# B&R Automation Studio project GAT (part 3)

### Alarm.mpalarmxcore - 5PPC2200_AL14_000/mappServices/Alarms/Alarm.mpalarmxcore
```
Element gAlarmXMpLink (Type=mpalarmxcore)
  mapp.AlarmX.Core:
    BySeverity:
      [0]:
        Severity = 1..9
        [0] = Reaction
          Name = Info
      [1]:
        Severity = 10..19
        [0] = Reaction
          Name = Warning
      [2]:
        Severity = 20..29
        [0] = Reaction
          Name = Error
  mapp.AlarmX.Core.Configuration:
    [0]:
      Name = EmergencyStop_0
      Message = {$Alarms/EmergencyStop.0}
      Severity = 29
      Behavior = DiscreteValueMonitoring
        Monitoring:
          MonitoredPV = ::AlarmMgt:SafetyInputs.EmergencyStop[0]
          TriggerValues:
            [0] = 1
    [1]:
      Name = EmergencyStop_1
      Message = {$Alarms/EmergencyStop.1}
      Behavior = DiscreteValueMonitoring
        Monitoring:
          MonitoredPV = ::AlarmMgt:SafetyInputs.EmergencyStop[1]
          TriggerValues:
            [0] = 1
    [2]:
      Name = EmergencyStop_2
      Message = {$Alarms/EmergencyStop.2}
      Behavior = DiscreteValueMonitoring
        Monitoring:
          MonitoredPV = ::AlarmMgt:SafetyInputs.EmergencyStop[2]
          TriggerValues:
            [0] = 1
    [3]:
      Name = SafetyDoor_0
      Message = {$Alarms/SafetyDoor.0}
      Severity = 29
      Behavior = DiscreteValueMonitoring
        Monitoring:
          MonitoredPV = ::AlarmMgt:SafetyInputs.SafetyDoor[0]
          TriggerValues:
            [0] = 1
    [4]:
      Name = SafetyDoor_1
      Message = {$Alarms/SafetyDoor.1}
      Severity = 29
      Behavior = DiscreteValueMonitoring
        Monitoring:
          MonitoredPV = ::AlarmMgt:SafetyInputs.SafetyDoor[1]
          TriggerValues:
            [0] = 1
    [5]:
      Name = SafetyDoor_2
      Message = {$Alarms/SafetyDoor.2}
      Severity = 29
      Behavior = DiscreteValueMonitoring
        Monitoring:
          MonitoredPV = ::AlarmMgt:SafetyInputs.SafetyDoor[2]
          TriggerValues:
            [0] = 1
    [6]:
      Name = SafetyDoor_3
      Message = {$Alarms/SafetyDoor.3}
      Severity = 29
      Behavior = DiscreteValueMonitoring
        Monitoring:
          MonitoredPV = ::AlarmMgt:SafetyInputs.SafetyDoor[3]
          TriggerValues:
            [0] = 1
    [7]:
      Name = SafetyDoor_4
      Message = {$Alarms/SafetyDoor.4}
      Severity = 29
      Behavior = DiscreteValueMonitoring
        Monitoring:
          MonitoredPV = ::AlarmMgt:SafetyInputs.SafetyDoor[4]
          TriggerValues:
            [0] = 1
    [8]:
      Name = SafetyDoor_5
      Message = {$Alarms/SafetyDoor.5}
      Severity = 29
      Behavior = DiscreteValueMonitoring
        Monitoring:
          MonitoredPV = ::AlarmMgt:SafetyInputs.SafetyDoor[5]
          TriggerValues:
            [0] = 1
    [9]:
      Name = LevelMonitoringExample
      Message = {$Alarms/LimitMonitoringExample} {=$Alarms/{$LimitText}}
      Behavior = LevelMonitoring
        Monitoring:
          MonitoredPV = ::AlarmMgt:AlarmExamples.LevelMonitoring
          LowLimitEnable = Static
            Limit = 20
            LimitText = LevelMonitoringAlarmLowTextExample
            LowLowLimitEnable = Static
              Limit = 10
              LimitText = LevelMonitoringAlarmLowLowTextExample
          HighLimitEnable = Static
            Limit = 80
            LimitText = LevelMonitoringAlarmHighTextExample
            HighHighLimitEnable = Static
              Limit = 90
              LimitText = LevelMonitoringAlarmHighHighTextExample
    [10]:
      Name = DeviationMonitoringExample
      Message = {$Alarms/LimitText}
      Behavior = DeviationMonitoring
        Monitoring:
          MonitoredPV = ::AlarmMgt:AlarmExamples.DeviationMonitoring
          SetpointPV = ::AlarmMgt:AlarmExamples.DeviationMonitoringSetpoint
          LowLimitEnable = Static
            Limit = -5
            LimitText = Low limit exceeded
          HighLimitEnable = Static
            Limit = 5
            LimitText = High limit exceeded
    [11]:
      Name = RateOfChangeExample
      Message = {$Alarms/RateOfChangeAlarmExample}
      Behavior = RateOfChangeMonitoring
        Monitoring:
          MonitoredPV = ::AlarmMgt:AlarmExamples.RateOfChange
          HighLimitEnable = Static
            Limit = 5
            LimitText = High limit exceeded
    [12]:
      Name = SnippetExample
      Message = {$Alarms/SnippetAlarmExample}
      Behavior = DiscreteValueMonitoring
        Monitoring:
          MonitoredPV = ::AlarmMgt:AlarmExamples.SnippetValue
          TriggerValues:
            [0] = 50..100
    [13]:
      Name = MpAlarmXControlExample
      Message = {$Alarms/Alarm.0}
      Severity = 20
      Behavior:
        Async = TRUE
    [14]:
      Name = Alarm0
      Message = {$Alarms/Alarm.0}
      Behavior = DiscreteValueMonitoring
        Monitoring:
          MonitoredPV = ::AlarmMgt:Alarms[0]
          InhibitPV = ::AlarmMgt:CommissioningModeActive
          TriggerValues:
            [0] = 1
    [15]:
      Name = Alarm1
      Message = {$Alarms/Alarm.1}
      Code = 1
      Behavior = DiscreteValueMonitoring
        Monitoring:
          MonitoredPV = ::AlarmMgt:Alarms[1]
          TriggerValues:
            [0] = 1
    [16]:
      Name = Alarm2
      Message = {$Alarms/Alarm.2}
      Code = 2
      Behavior = DiscreteValueMonitoring
        Monitoring:
          MonitoredPV = ::AlarmMgt:Alarms[2]
          TriggerValues:
            [0] = 1
    [17]:
      Name = Alarm3
      Message = {$Alarms/Alarm.3}
      Code = 3
      Behavior = DiscreteValueMonitoring
        Monitoring:
          MonitoredPV = ::AlarmMgt:Alarms[3]
          TriggerValues:
            [0] = 1
    [18]:
      Name = Alarm4
      Message = {$Alarms/Alarm.4}
      Code = 4
      Behavior = DiscreteValueMonitoring
        Monitoring:
          MonitoredPV = ::AlarmMgt:Alarms[4]
          TriggerValues:
            [0] = 1
    [19]:
      Name = Alarm5
      Message = {$Alarms/Alarm.5}
      Code = 5
      Behavior = DiscreteValueMonitoring
        Monitoring:
          MonitoredPV = ::AlarmMgt:Alarms[5]
          TriggerValues:
            [0] = 1
    [20]:
      Name = Alarm6
      Message = {$Alarms/Alarm.6}
      Code = 6
      Behavior = DiscreteValueMonitoring
        Monitoring:
          MonitoredPV = ::AlarmMgt:Alarms[6]
          TriggerValues:
            [0] = 1
    [21]:
      Name = Alarm7
      Message = {$Alarms/Alarm.7}
      Code = 7
      Behavior = DiscreteValueMonitoring
        Monitoring:
          MonitoredPV = ::AlarmMgt:Alarms[7]
          TriggerValues:
            [0] = 1
    [22]:
      Name = Alarm8
      Message = {$Alarms/Alarm.8}
      Code = 8
      Behavior = DiscreteValueMonitoring
        Monitoring:
          MonitoredPV = ::AlarmMgt:Alarms[8]
          TriggerValues:
            [0] = 1
    [23]:
      Name = Alarm9
      Message = {$Alarms/Alarm.9}
      Code = 9
      Behavior = DiscreteValueMonitoring
        Monitoring:
          MonitoredPV = ::AlarmMgt:Alarms[9]
          TriggerValues:
            [0] = 1
    [24]:
      Name = Alarm10
      Message = {$Alarms/Alarm.10}
      Code = 10
      Behavior = DiscreteValueMonitoring
        Monitoring:
          MonitoredPV = ::AlarmMgt:Alarms[10]
          TriggerValues:
            [0] = 1
    [25]:
      Name = Alarm11
      Message = {$Alarms/Alarm.11}
      Code = 11
      Behavior = DiscreteValueMonitoring
        Monitoring:
          MonitoredPV = ::AlarmMgt:Alarms[11]
          TriggerValues:
            [0] = 1
    [26]:
      Name = Alarm12
      Message = {$Alarms/Alarm.12}
      Code = 12
      Behavior = DiscreteValueMonitoring
        Monitoring:
          MonitoredPV = ::AlarmMgt:Alarms[12]
          TriggerValues:
            [0] = 1
    [27]:
      Name = Alarm13
      Message = {$Alarms/Alarm.13}
      Code = 13
      Behavior = DiscreteValueMonitoring
        Monitoring:
          MonitoredPV = ::AlarmMgt:Alarms[13]
          TriggerValues:
            [0] = 1
    [28]:
      Name = Alarm14
      Message = {$Alarms/Alarm.14}
      Code = 14
      Behavior = DiscreteValueMonitoring
        Monitoring:
          MonitoredPV = ::AlarmMgt:Alarms[14]
          TriggerValues:
            [0] = 1
    [29]:
      Name = Alarm15
      Message = {$Alarms/Alarm.15}
      Code = 15
      Behavior = DiscreteValueMonitoring
        Monitoring:
          MonitoredPV = ::AlarmMgt:Alarms[15]
          TriggerValues:
            [0] = 1
    [30]:
      Name = Alarm16
      Message = {$Alarms/Alarm.16}
      Code = 16
      Behavior = DiscreteValueMonitoring
        Monitoring:
          MonitoredPV = ::AlarmMgt:Alarms[16]
          TriggerValues:
            [0] = 1
    [31]:
      Name = Alarm17
      Message = {$Alarms/Alarm.17}
      Code = 17
      Behavior = DiscreteValueMonitoring
        Monitoring:
          MonitoredPV = ::AlarmMgt:Alarms[17]
          TriggerValues:
            [0] = 1
    [32]:
      Name = Alarm18
      Message = {$Alarms/Alarm.18}
      Code = 18
      Behavior = DiscreteValueMonitoring
        Monitoring:
          MonitoredPV = ::AlarmMgt:Alarms[18]
          TriggerValues:
            [0] = 1
    [33]:
      Name = Alarm19
      Message = {$Alarms/Alarm.19}
      Code = 19
      Behavior = DiscreteValueMonitoring
        Monitoring:
          MonitoredPV = ::AlarmMgt:Alarms[19]
          TriggerValues:
            [0] = 1
    [34]:
      Name = Alarm20
      Message = {$Alarms/Alarm.20}
      Behavior = DiscreteValueMonitoring
        Monitoring:
          MonitoredPV = ::AlarmMgt:Alarms[20]
          TriggerValues:
            [0] = 1
    [35]:
      Name = Alarm21
      Message = {$Alarms/Alarm.21}
      Code = 21
      Behavior = DiscreteValueMonitoring
        Monitoring:
          MonitoredPV = ::AlarmMgt:Alarms[21]
          TriggerValues:
            [0] = 1
    [36]:
      Name = Alarm22
      Message = {$Alarms/Alarm.22}
      Code = 22
      Behavior = DiscreteValueMonitoring
        Monitoring:
          MonitoredPV = ::AlarmMgt:Alarms[22]
          TriggerValues:
            [0] = 1
    [37]:
      Name = Alarm23
      Message = {$Alarms/Alarm.23}
      Code = 23
      Behavior = DiscreteValueMonitoring
        Monitoring:
          MonitoredPV = ::AlarmMgt:Alarms[23]
          TriggerValues:
            [0] = 1
    [38]:
      Name = Alarm24
      Message = {$Alarms/Alarm.24}
      Code = 24
      Behavior = DiscreteValueMonitoring
        Monitoring:
          MonitoredPV = ::AlarmMgt:Alarms[24]
          TriggerValues:
            [0] = 1
    [39]:
      Name = Alarm25
      Message = {$Alarms/Alarm.25}
      Code = 25
      Behavior = DiscreteValueMonitoring
        Monitoring:
          MonitoredPV = ::AlarmMgt:Alarms[25]
          TriggerValues:
            [0] = 1
    [40]:
      Name = Alarm26
      Message = {$Alarms/Alarm.26}
      Code = 26
      Behavior = DiscreteValueMonitoring
        Monitoring:
          MonitoredPV = ::AlarmMgt:Alarms[26]
          TriggerValues:
            [0] = 1
    [41]:
      Name = Alarm27
      Message = {$Alarms/Alarm.27}
      Code = 27
      Behavior = DiscreteValueMonitoring
        Monitoring:
          MonitoredPV = ::AlarmMgt:Alarms[27]
          TriggerValues:
            [0] = 1
    [42]:
      Name = Alarm28
      Message = {$Alarms/Alarm.28}
      Code = 28
      Behavior = DiscreteValueMonitoring
        Monitoring:
          MonitoredPV = ::AlarmMgt:Alarms[28]
          TriggerValues:
            [0] = 1
    [43]:
      Name = Alarm29
      Message = {$Alarms/Alarm.29}
      Code = 29
      Behavior = DiscreteValueMonitoring
        Monitoring:
          MonitoredPV = ::AlarmMgt:Alarms[29]
          TriggerValues:
            [0] = 1
    [44]:
      Name = Alarm30
      Message = {$Alarms/Alarm.30}
      Behavior = DiscreteValueMonitoring
        Monitoring:
          MonitoredPV = ::AlarmMgt:Alarms[30]
          TriggerValues:
            [0] = 1
    [45]:
      Name = Alarm31
      Message = {$Alarms/Alarm.31}
      Code = 31
      Behavior = DiscreteValueMonitoring
        Monitoring:
          MonitoredPV = ::AlarmMgt:Alarms[31]
          TriggerValues:
            [0] = 1
    [46]:
      Name = Alarm32
      Message = {$Alarms/Alarm.32}
      Code = 32
      Behavior = DiscreteValueMonitoring
        Monitoring:
          MonitoredPV = ::AlarmMgt:Alarms[32]
          TriggerValues:
            [0] = 1
    [47]:
      Name = Alarm33
      Message = {$Alarms/Alarm.33}
      Code = 33
      Behavior = DiscreteValueMonitoring
        Monitoring:
          MonitoredPV = ::AlarmMgt:Alarms[33]
          TriggerValues:
            [0] = 1
    [48]:
      Name = Alarm34
      Message = {$Alarms/Alarm.34}
      Code = 34
      Behavior = DiscreteValueMonitoring
        Monitoring:
          MonitoredPV = ::AlarmMgt:Alarms[34]
          TriggerValues:
            [0] = 1
    [49]:
      Name = Alarm35
      Message = {$Alarms/Alarm.35}
      Code = 35
      Behavior = DiscreteValueMonitoring
        Monitoring:
          MonitoredPV = ::AlarmMgt:Alarms[35]
          TriggerValues:
            [0] = 1
    [50]:
      Name = Alarm36
      Message = {$Alarms/Alarm.36}
      Code = 36
      Behavior = DiscreteValueMonitoring
        Monitoring:
          MonitoredPV = ::AlarmMgt:Alarms[36]
          TriggerValues:
            [0] = 1
    [51]:
      Name = Alarm37
      Message = {$Alarms/Alarm.37}
      Code = 37
      Behavior = DiscreteValueMonitoring
        Monitoring:
          MonitoredPV = ::AlarmMgt:Alarms[37]
          TriggerValues:
            [0] = 1
    [52]:
      Name = Alarm38
      Message = {$Alarms/Alarm.38}
      Code = 38
      Behavior = DiscreteValueMonitoring
        Monitoring:
          MonitoredPV = ::AlarmMgt:Alarms[38]
          TriggerValues:
            [0] = 1
    [53]:
      Name = Alarm39
      Message = {$Alarms/Alarm.39}
      Code = 39
      Behavior = DiscreteValueMonitoring
        Monitoring:
          MonitoredPV = ::AlarmMgt:Alarms[39]
          TriggerValues:
            [0] = 1
    [54]:
      Name = Alarm40
      Message = {$Alarms/Alarm.40}
      Behavior = DiscreteValueMonitoring
        Monitoring:
          MonitoredPV = ::AlarmMgt:Alarms[40]
          TriggerValues:
            [0] = 1
    [55]:
      Name = Alarm41
      Message = {$Alarms/Alarm.41}
      Code = 41
      Behavior = DiscreteValueMonitoring
        Monitoring:
          MonitoredPV = ::AlarmMgt:Alarms[41]
          TriggerValues:
            [0] = 1
    [56]:
      Name = Alarm42
      Message = {$Alarms/Alarm.42}
      Code = 42
      Behavior = DiscreteValueMonitoring
        Monitoring:
          MonitoredPV = ::AlarmMgt:Alarms[42]
          TriggerValues:
            [0] = 1
    [57]:
      Name = Alarm43
      Message = {$Alarms/Alarm.43}
      Code = 43
      Behavior = DiscreteValueMonitoring
        Monitoring:
          MonitoredPV = ::AlarmMgt:Alarms[43]
          TriggerValues:
            [0] = 1
    [58]:
      Name = Alarm44
      Message = {$Alarms/Alarm.44}
      Code = 44
      Behavior = DiscreteValueMonitoring
        Monitoring:
          MonitoredPV = ::AlarmMgt:Alarms[44]
          TriggerValues:
            [0] = 1
    [59]:
      Name = Alarm45
      Message = {$Alarms/Alarm.45}
      Code = 45
      Behavior = DiscreteValueMonitoring
        Monitoring:
          MonitoredPV = ::AlarmMgt:Alarms[45]
          TriggerValues:
            [0] = 1
    [60]:
      Name = Alarm46
      Message = {$Alarms/Alarm.46}
      Code = 46
      Behavior = DiscreteValueMonitoring
        Monitoring:
          MonitoredPV = ::AlarmMgt:Alarms[46]
          TriggerValues:
            [0] = 1
    [61]:
      Name = Alarm47
      Message = {$Alarms/Alarm.47}
      Code = 47
      Behavior = DiscreteValueMonitoring
        Monitoring:
          MonitoredPV = ::AlarmMgt:Alarms[47]
          TriggerValues:
            [0] = 1
    [62]:
      Name = Alarm48
      Message = {$Alarms/Alarm.48}
      Code = 48
      Behavior = DiscreteValueMonitoring
        Monitoring:
          MonitoredPV = ::AlarmMgt:Alarms[48]
          TriggerValues:
            [0] = 1
    [63]:
      Name = Alarm49
      Message = {$Alarms/Alarm.49}
      Code = 49
      Behavior = DiscreteValueMonitoring
        Monitoring:
          MonitoredPV = ::AlarmMgt:Alarms[49]
          TriggerValues:
            [0] = 1
    [64]:
      Name = Alarm50
      Message = {$Alarms/Alarm.50}
      Behavior = DiscreteValueMonitoring
        Monitoring:
          MonitoredPV = ::AlarmMgt:Alarms[50]
          TriggerValues:
            [0] = 1
    [65]:
      Name = Alarm51
      Message = {$Alarms/Alarm.51}
      Code = 51
      Behavior = DiscreteValueMonitoring
        Monitoring:
          MonitoredPV = ::AlarmMgt:Alarms[51]
          TriggerValues:
            [0] = 1
    [66]:
      Name = Alarm52
      Message = {$Alarms/Alarm.52}
      Code = 52
      Behavior = DiscreteValueMonitoring
        Monitoring:
          MonitoredPV = ::AlarmMgt:Alarms[52]
          TriggerValues:
            [0] = 1
    [67]:
      Name = Alarm53
      Message = {$Alarms/Alarm.53}
      Code = 53
      Behavior = DiscreteValueMonitoring
        Monitoring:
          MonitoredPV = ::AlarmMgt:Alarms[53]
          TriggerValues:
            [0] = 1
    [68]:
      Name = Alarm54
      Message = {$Alarms/Alarm.54}
      Code = 54
      Behavior = DiscreteValueMonitoring
        Monitoring:
          MonitoredPV = ::AlarmMgt:Alarms[54]
          TriggerValues:
            [0] = 1
    [69]:
      Name = Alarm55
      Message = {$Alarms/Alarm.55}
      Code = 55
      Behavior = DiscreteValueMonitoring
        Monitoring:
          MonitoredPV = ::AlarmMgt:Alarms[55]
          TriggerValues:
            [0] = 1
    [70]:
      Name = Alarm56
      Message = {$Alarms/Alarm.56}
      Code = 56
      Behavior = DiscreteValueMonitoring
        Monitoring:
          MonitoredPV = ::AlarmMgt:Alarms[56]
          TriggerValues:
            [0] = 1
    [71]:
      Name = Alarm57
      Message = {$Alarms/Alarm.57}
      Code = 57
      Behavior = DiscreteValueMonitoring
        Monitoring:
          MonitoredPV = ::AlarmMgt:Alarms[57]
          TriggerValues:
            [0] = 1
    [72]:
      Name = Alarm58
      Message = {$Alarms/Alarm.58}
      Code = 58
      Behavior = DiscreteValueMonitoring
        Monitoring:
          MonitoredPV = ::AlarmMgt:Alarms[58]
          TriggerValues:
            [0] = 1
    [73]:
      Name = Alarm59
      Message = {$Alarms/Alarm.59}
      Code = 59
      Behavior = DiscreteValueMonitoring
        Monitoring:
          MonitoredPV = ::AlarmMgt:Alarms[59]
          TriggerValues:
            [0] = 1
    [74]:
      Name = Alarm60
      Message = {$Alarms/Alarm.60}
      Behavior = DiscreteValueMonitoring
        Monitoring:
          MonitoredPV = ::AlarmMgt:Alarms[60]
          TriggerValues:
            [0] = 1
    [75]:
      Name = Alarm61
      Message = {$Alarms/Alarm.61}
      Code = 61
      Behavior = DiscreteValueMonitoring
        Monitoring:
          MonitoredPV = ::AlarmMgt:Alarms[61]
          TriggerValues:
            [0] = 1
    [76]:
      Name = Alarm62
      Message = {$Alarms/Alarm.62}
      Code = 62
      Behavior = DiscreteValueMonitoring
        Monitoring:
          MonitoredPV = ::AlarmMgt:Alarms[62]
          TriggerValues:
            [0] = 1
    [77]:
      Name = Alarm63
      Message = {$Alarms/Alarm.63}
      Code = 63
      Behavior = DiscreteValueMonitoring
        Monitoring:
          MonitoredPV = ::AlarmMgt:Alarms[63]
          TriggerValues:
            [0] = 1
    [78]:
      Name = Alarm64
      Message = {$Alarms/Alarm.64}
      Code = 64
      Behavior = DiscreteValueMonitoring
        Monitoring:
          MonitoredPV = ::AlarmMgt:Alarms[64]
          TriggerValues:
            [0] = 1
    [79]:
      Name = Alarm65
      Message = {$Alarms/Alarm.65}
      Code = 65
      Behavior = DiscreteValueMonitoring
        Monitoring:
          MonitoredPV = ::AlarmMgt:Alarms[65]
          TriggerValues:
            [0] = 1
    [80]:
      Name = Alarm66
      Message = {$Alarms/Alarm.66}
      Code = 66
      Behavior = DiscreteValueMonitoring
        Monitoring:
          MonitoredPV = ::AlarmMgt:Alarms[66]
          TriggerValues:
            [0] = 1
    [81]:
      Name = Alarm67
      Message = {$Alarms/Alarm.67}
      Code = 67
      Behavior = DiscreteValueMonitoring
        Monitoring:
          MonitoredPV = ::AlarmMgt:Alarms[67]
          TriggerValues:
            [0] = 1
    [82]:
      Name = Alarm68
      Message = {$Alarms/Alarm.68}
      Code = 68
      Behavior = DiscreteValueMonitoring
        Monitoring:
          MonitoredPV = ::AlarmMgt:Alarms[68]
          TriggerValues:
            [0] = 1
    [83]:
      Name = Alarm69
      Message = {$Alarms/Alarm.69}
      Code = 69
      Behavior = DiscreteValueMonitoring
        Monitoring:
          MonitoredPV = ::AlarmMgt:Alarms[69]
          TriggerValues:
            [0] = 1
    [84]:
      Name = Alarm70
      Message = {$Alarms/Alarm.70}
      Behavior = DiscreteValueMonitoring
        Monitoring:
          MonitoredPV = ::AlarmMgt:Alarms[70]
          TriggerValues:
            [0] = 1
    [85]:
      Name = Alarm71
      Message = {$Alarms/Alarm.71}
      Code = 71
      Behavior = DiscreteValueMonitoring
        Monitoring:
          MonitoredPV = ::AlarmMgt:Alarms[71]
          TriggerValues:
            [0] = 1
    [86]:
      Name = Alarm72
      Message = {$Alarms/Alarm.72}
      Code = 72
      Behavior = DiscreteValueMonitoring
        Monitoring:
          MonitoredPV = ::AlarmMgt:Alarms[72]
          TriggerValues:
            [0] = 1
    [87]:
      Name = Alarm73
      Message = {$Alarms/Alarm.73}
      Code = 73
      Behavior = DiscreteValueMonitoring
        Monitoring:
          MonitoredPV = ::AlarmMgt:Alarms[73]
          TriggerValues:
            [0] = 1
    [88]:
      Name = Alarm74
      Message = {$Alarms/Alarm.74}
      Code = 74
      Behavior = DiscreteValueMonitoring
        Monitoring:
          MonitoredPV = ::AlarmMgt:Alarms[74]
          TriggerValues:
            [0] = 1
    [89]:
      Name = Alarm75
      Message = {$Alarms/Alarm.75}
      Code = 75
      Behavior = DiscreteValueMonitoring
        Monitoring:
          MonitoredPV = ::AlarmMgt:Alarms[75]
          TriggerValues:
            [0] = 1
    [90]:
      Name = Alarm76
      Message = {$Alarms/Alarm.76}
      Code = 76
      Behavior = DiscreteValueMonitoring
        Monitoring:
          MonitoredPV = ::AlarmMgt:Alarms[76]
          TriggerValues:
            [0] = 1
    [91]:
      Name = Alarm77
      Message = {$Alarms/Alarm.77}
      Code = 77
      Behavior = DiscreteValueMonitoring
        Monitoring:
          MonitoredPV = ::AlarmMgt:Alarms[77]
          TriggerValues:
            [0] = 1
    [92]:
      Name = Alarm78
      Message = {$Alarms/Alarm.78}
      Code = 78
      Behavior = DiscreteValueMonitoring
        Monitoring:
          MonitoredPV = ::AlarmMgt:Alarms[78]
          TriggerValues:
            [0] = 1
    [93]:
      Name = Alarm79
      Message = {$Alarms/Alarm.79}
      Code = 79
      Behavior = DiscreteValueMonitoring
        Monitoring:
          MonitoredPV = ::AlarmMgt:Alarms[79]
          TriggerValues:
            [0] = 1
    [94]:
      Name = Alarm80
      Message = {$Alarms/Alarm.80}
      Behavior = DiscreteValueMonitoring
        Monitoring:
          MonitoredPV = ::AlarmMgt:Alarms[80]
          TriggerValues:
            [0] = 1
    [95]:
      Name = Alarm81
      Message = {$Alarms/Alarm.81}
      Code = 81
      Behavior = DiscreteValueMonitoring
        Monitoring:
          MonitoredPV = ::AlarmMgt:Alarms[81]
          TriggerValues:
            [0] = 1
    [96]:
      Name = Alarm82
      Message = {$Alarms/Alarm.82}
      Code = 82
      Behavior = DiscreteValueMonitoring
        Monitoring:
          MonitoredPV = ::AlarmMgt:Alarms[82]
          TriggerValues:
            [0] = 1
    [97]:
      Name = Alarm83
      Message = {$Alarms/Alarm.83}
      Code = 83
      Behavior = DiscreteValueMonitoring
        Monitoring:
          MonitoredPV = ::AlarmMgt:Alarms[83]
          TriggerValues:
            [0] = 1
    [98]:
      Name = Alarm84
      Message = {$Alarms/Alarm.84}
      Code = 84
      Behavior = DiscreteValueMonitoring
        Monitoring:
          MonitoredPV = ::AlarmMgt:Alarms[84]
          TriggerValues:
            [0] = 1
    [99]:
      Name = Alarm85
      Message = {$Alarms/Alarm.85}
      Code = 85
      Behavior = DiscreteValueMonitoring
        Monitoring:
          MonitoredPV = ::AlarmMgt:Alarms[85]
          TriggerValues:
            [0] = 1
    [100]:
      Name = Alarm86
      Message = {$Alarms/Alarm.86}
      Code = 86
      Behavior = DiscreteValueMonitoring
        Monitoring:
          MonitoredPV = ::AlarmMgt:Alarms[86]
          TriggerValues:
            [0] = 1
    [101]:
      Name = Alarm87
      Message = {$Alarms/Alarm.87}
      Code = 87
      Behavior = DiscreteValueMonitoring
        Monitoring:
          MonitoredPV = ::AlarmMgt:Alarms[87]
          TriggerValues:
            [0] = 1
    [102]:
      Name = Alarm88
      Message = {$Alarms/Alarm.88}
      Code = 88
      Behavior = DiscreteValueMonitoring
        Monitoring:
          MonitoredPV = ::AlarmMgt:Alarms[88]
          TriggerValues:
            [0] = 1
    [103]:
      Name = Alarm89
      Message = {$Alarms/Alarm.89}
      Code = 89
      Behavior = DiscreteValueMonitoring
        Monitoring:
          MonitoredPV = ::AlarmMgt:Alarms[89]
          TriggerValues:
            [0] = 1
    [104]:
      Name = Alarm90
      Message = {$Alarms/Alarm.90}
      Behavior = DiscreteValueMonitoring
        Monitoring:
          MonitoredPV = ::AlarmMgt:Alarms[90]
          TriggerValues:
            [0] = 1
    [105]:
      Name = Alarm91
      Message = {$Alarms/Alarm.91}
      Code = 91
      Behavior = DiscreteValueMonitoring
        Monitoring:
          MonitoredPV = ::AlarmMgt:Alarms[91]
          TriggerValues:
            [0] = 1
    [106]:
      Name = Alarm92
      Message = {$Alarms/Alarm.92}
      Code = 92
      Behavior = DiscreteValueMonitoring
        Monitoring:
          MonitoredPV = ::AlarmMgt:Alarms[92]
          TriggerValues:
            [0] = 1
    [107]:
      Name = Alarm93
      Message = {$Alarms/Alarm.93}
      Code = 93
      Behavior = DiscreteValueMonitoring
        Monitoring:
          MonitoredPV = ::AlarmMgt:Alarms[93]
          TriggerValues:
            [0] = 1
    [108]:
      Name = Alarm94
      Message = {$Alarms/Alarm.94}
      Code = 94
      Behavior = DiscreteValueMonitoring
        Monitoring:
          MonitoredPV = ::AlarmMgt:Alarms[94]
          TriggerValues:
            [0] = 1
    [109]:
      Name = Alarm95
      Message = {$Alarms/Alarm.95}
      Code = 95
      Behavior = DiscreteValueMonitoring
        Monitoring:
          MonitoredPV = ::AlarmMgt:Alarms[95]
          TriggerValues:
            [0] = 1
    [110]:
      Name = Alarm96
      Message = {$Alarms/Alarm.96}
      Code = 96
      Behavior = DiscreteValueMonitoring
        Monitoring:
          MonitoredPV = ::AlarmMgt:Alarms[96]
          TriggerValues:
            [0] = 1
    [111]:
      Name = Alarm97
      Message = {$Alarms/Alarm.97}
      Code = 97
      Behavior = DiscreteValueMonitoring
        Monitoring:
          MonitoredPV = ::AlarmMgt:Alarms[97]
          TriggerValues:
            [0] = 1
    [112]:
      Name = Alarm98
      Message = {$Alarms/Alarm.98}
      Code = 98
      Behavior = DiscreteValueMonitoring
        Monitoring:
          MonitoredPV = ::AlarmMgt:Alarms[98]
          TriggerValues:
            [0] = 1
    [113]:
      Name = Alarm99
      Message = {$Alarms/Alarm.99}
      Code = 99
      Behavior = DiscreteValueMonitoring
        Monitoring:
          MonitoredPV = ::AlarmMgt:Alarms[99]
          TriggerValues:
            [0] = 1
  mapp.AlarmX.Core.Snippets:
    AutoDetect = 1
    [0]:
      Key = snippet1
      Value:
        PV = ::AlarmMgt:AlarmExamples.SnippetValue
  mapp.AlarmX.Core.Queries:
    [0]:
      Name = ActiveAlarms
      Update = ::AlarmMgt:AlarmQuery.ActiveAlarmUpdateCount
      Source:
        SELECT:
          [0]:
            PV = ::AlarmMgt:AlarmQuery.Alarms[].Name
          [1]:
            Column = Message
            PV = ::AlarmMgt:AlarmQuery.Alarms[].Message
          [2]:
            Column = Code
            PV = ::AlarmMgt:AlarmQuery.Alarms[].Code
          [3]:
            Column = Severity
            PV = ::AlarmMgt:AlarmQuery.Alarms[].Severity
          [4]:
            Column = Scope
            PV = ::AlarmMgt:AlarmQuery.Alarms[].Scope
          [5]:
            Column = TimeStamp
            PV = ::AlarmMgt:AlarmQuery.Alarms[].TimeStamp
          [6]:
            Column = AdditionalInformation1
            PV = ::AlarmMgt:AlarmQuery.Alarms[].AdditionalInfo
          [7]:
            Column = StateActive
            PV = ::AlarmMgt:AlarmQuery.Alarms[].Active
          [8]:
            Column = StateAcknowledged
            PV = ::AlarmMgt:AlarmQuery.Alarms[].Acknowledged
```

### Axis1Alm.mpalarmxcore - 5PPC2200_AL14_000/mappServices/AppAxis_1/Axis1Alm.mpalarmxcore
```
Element gMpLinkAlarmXCoreAppAxis_1 (Type=mpalarmxcore)
  mapp.AlarmX.Core:
    BySeverity:
      [0]:
        Severity = 1..9
        [0] = Reaction
          Name = Info
        [1] = Escalate
        [2] = Remain
      [1]:
        Severity = 10..19
        [0] = Reaction
          Name = Warning
        [1] = Escalate
        [2] = Remain
      [2]:
        Severity = 20..29
        [0] = Reaction
          Name = Error
        [1] = Escalate
        [2] = Remain
    Default:
      [0] = Reaction
        Name = Duplicate
      [1] = Escalate
      [2] = Remain
  mapp.AlarmX.Core.Configuration:
    [0]:
      Name = ReferenceRequired
      Message = {$IAT/AppAxis_1/Info/Name} : {$Axis/Alarms/ReferenceRequired}
      Severity = 10
      Behavior = DiscreteValueMonitoring
        Monitoring:
          MonitoredPV = ::AppAxis_1:AxisControl.Status.ReferenceRequired
          TriggerValues:
            [0] = 1
    [1]:
      Name = AppAxis_1SpeedNotSet
      Message = {$IAT/AppAxis_1/Info/Name} : {$Axis/Alarms/AppAxis_1SpeedNotSet}
      Code = 250
      Severity = 20
      Behavior:
        Async = TRUE
  mapp.AlarmX.Core.Snippets:
    [0]:
      Key = AppAxis_1Speed
      Value:
        PV = ::AppAxis_1:AxisControl.Parameters.Velocity
```

### Axis1Grp.mpcomgroup - 5PPC2200_AL14_000/mappServices/AppAxis_1/Axis1Grp.mpcomgroup
```
Element gGroupAppAxis_1 (Type=mpcomgroup)
  Linking:
    Subnodes:
      0 = gAppAxis_1
      1 = gAlarmXCore_AppAxis_1
  Alarms = MpAlarmX
```

### AuditCfg.mpaudittrail - 5PPC2200_AL14_000/mappServices/Audit/AuditCfg.mpaudittrail
```
Element gAuditTrailMpLink (Type=mpaudittrail)
  Audit:
    Events:
      [0] = 19
      [1] = 2
      [2] = 48
      [3] = 18
      [4] = 33
    TextSource = TXT
      Name = 
      OutputFormat = EventLog/Root
    Archive = On
    Export:
      FileType = 2
      Encrypt = FALSE
      PDF:
        DefaultFont = 3
  Alarms = MpAlarmX
```

### AuditFile.mpfilemanagerui - 5PPC2200_AL14_000/mappServices/Audit/AuditFile.mpfilemanagerui
```
Element gMpLinkFileManagerUIAudit (Type=mpfilemanagerui)
  Alarms = MpAlarmX
    mapp.AlarmX.Core.Configuration:
      [0]:
        Message = {$File/Alarms/DeviceNotFound}
      [1]:
        Message = {$File/Alarms/AlreadyExisting}
      [2]:
        Message = {$File/Alarms/FileSystemError}
```

### Backup.mpbackupcore - 5PPC2200_AL14_000/mappServices/Backup/Backup.mpbackupcore
```
Element gMpLinkBackupCore (Type=mpbackupcore)
  Backup:
    AutomaticBackup = Enabled
      Mode = Weekly
      OverwriteOldest = Enabled
        MaximumNumberOfBackups = 5
    AutomaticUpdate = Notify
      DeviceName = mappBackup
  Alarms = MpAlarmX
```

### BackupCfg.mpbackupcore - 5PPC2200_AL14_000/mappServices/Backup/BackupCfg.mpbackupcore
```
Element gMpLinkBackupCore (Type=mpbackupcore)
  Backup:
    AutomaticBackup = Enabled
      Mode = Weekly
      OverwriteOldest = Enabled
        MaximumNumberOfBackups = 5
    AutomaticUpdate = Notify
      DeviceName = mappBackupFiles
  Alarms = MpAlarmX
```

### BackupFile.mpfilemanagerui - 5PPC2200_AL14_000/mappServices/Backup/BackupFile.mpfilemanagerui
```
Element gMpLinkFileManagerUIBackup (Type=mpfilemanagerui)
  Alarms = MpAlarmX
```

### ConvAlm.mpalarmxcore - 5PPC2200_AL14_000/mappServices/Conveyor/ConvAlm.mpalarmxcore
```
Element gAlarmXCore_Conveyor (Type=mpalarmxcore)
  mapp.AlarmX.Core:
    BySeverity:
      [0]:
        Severity = 1..9
        [0] = Reaction
          Name = Info
        [1] = Escalate
        [2] = Remain
      [1]:
        Severity = 10..19
        [0] = Reaction
          Name = Warning
        [1] = Escalate
        [2] = Remain
      [2]:
        Severity = 20..29
        [0] = Reaction
          Name = Error
        [1] = Escalate
        [2] = Remain
    Default:
      [0] = Reaction
        Name = Duplicate
      [1] = Escalate
      [2] = Remain
  mapp.AlarmX.Core.Configuration:
    [0]:
      Name = ReferenceRequired
      Message = {$IAT/Conveyor/Info/Name} : {$Conveyor/Alarms/ReferenceRequired}
      Severity = 10
      Behavior = DiscreteValueMonitoring
        Monitoring:
          MonitoredPV = ::Conveyor:AxisControl.Status.ReferenceRequired
          TriggerValues:
            [0] = 1
    [1]:
      Name = ConveyorSpeedNotSet
      Message = {$IAT/Conveyor/Alarms/ConveyorSpeedNotSet}
      Code = 250
      Severity = 20
      Behavior:
        Async = TRUE
  mapp.AlarmX.Core.Snippets:
    [0]:
      Key = ConveyorSpeed
      Value:
        PV = ::Conveyor:AxisControl.Parameters.Velocity
```

### ConvGrp.mpcomgroup - 5PPC2200_AL14_000/mappServices/Conveyor/ConvGrp.mpcomgroup
```
Element gGroupAppAxis_1 (Type=mpcomgroup)
  Linking:
    Subnodes:
      0 = gAxisAppAxis_1
      1 = gAlarmXCore_AppAxis_1
  Alarms = MpAlarmX
```

### CutterAlm.mpalarmxcore - 5PPC2200_AL14_000/mappServices/CrossCutter/CutterAlm.mpalarmxcore
```
Element gAlarmXCore_Cutter (Type=mpalarmxcore)
  mapp.AlarmX.Core:
    BySeverity:
      [0]:
        Severity = 1..9
        [0] = Reaction
          Name = Info
        [1] = Escalate
        [2] = Remain
      [1]:
        Severity = 10..19
        [0] = Reaction
          Name = Warning
        [1] = Escalate
        [2] = Remain
      [2]:
        Severity = 20..29
        [0] = Reaction
          Name = Error
        [1] = Escalate
        [2] = Remain
    Default:
      [0] = Reaction
        Name = Duplicate
      [1] = Escalate
      [2] = Remain
```

### DataCfg.mpdatarecorder - 5PPC2200_AL14_000/mappServices/Data/DataCfg.mpdatarecorder
```
Element gMpLinkDataRecorder (Type=mpdatarecorder)
  DataRecorder:
    MaxFileSize = 10000
    SaveInterval = 2000
    Format = PDF
      Font = 3
      OwnerPassword = 
      AllowCopy = TRUE
      AllowEdit = TRUE
    UnitDefinition = MeasurementSystemBased
      UnitDisplay = 1
  Alarms = MpAlarmX
```

### DataFile.mpfilemanagerui - 5PPC2200_AL14_000/mappServices/Data/DataFile.mpfilemanagerui
```
Element gMpLinkFileManagerUIData (Type=mpfilemanagerui)
  Alarms = MpAlarmX
    mapp.AlarmX.Core.Configuration:
      [0]:
        Message = {$File/Alarms/DeviceNotFound}
      [1]:
        Message = {$File/Alarms/AlreadyExisting}
      [2]:
        Message = {$File/Alarms/FileSystemError}
```

### FileMgr.mpfilemanagerui - 5PPC2200_AL14_000/mappServices/File/FileMgr.mpfilemanagerui
```
Element gMpLinkFileManagerUIData (Type=mpfilemanagerui)
  Alarms = MpAlarmX
    mapp.AlarmX.Core.Configuration:
      [0]:
        Message = {$File/Alarms/DeviceNotFound}
      [1]:
        Message = {$File/Alarms/AlreadyExisting}
      [2]:
        Message = {$File/Alarms/FileSystemError}
Element gMpLinkFileManagerUIReport (Type=mpfilemanagerui)
  Alarms = MpAlarmX
    mapp.AlarmX.Core.Configuration:
      [0]:
        Message = {$File/Alarms/DeviceNotFound}
      [1]:
        Message = {$File/Alarms/AlreadyExisting}
      [2]:
        Message = {$File/Alarms/FileSystemError}
Element gMpLinkFileManagerUIAudit (Type=mpfilemanagerui)
  Alarms = MpAlarmX
    mapp.AlarmX.Core.Configuration:
      [0]:
        Message = {$File/Alarms/DeviceNotFound}
      [1]:
        Message = {$File/Alarms/AlreadyExisting}
      [2]:
        Message = {$File/Alarms/FileSystemError}
Element gMpLinkFileManagerUIFile (Type=mpfilemanagerui)
  Alarms = MpAlarmX
    mapp.AlarmX.Core.Configuration:
      [0]:
        Message = {$File/Alarms/DeviceNotFound}
      [1]:
        Message = {$File/Alarms/AlreadyExisting}
      [2]:
        Message = {$File/Alarms/FileSystemError}
```

### MachineGrp.mpcomgroup - 5PPC2200_AL14_000/mappServices/MachineGrp.mpcomgroup
```
Element gMpLinkGroup (Type=mpcomgroup)
  Linking:
    Subnodes:
      0 = gMpLinkGroupAppAxis_1
      1 = gMpLinkAlarmXCore
      2 = gMpLinkRecipeXml
      3 = gMpLinkBackupCore
  Alarms = MpAlarmX
```

### Rcp.mprecipexml - 5PPC2200_AL14_000/mappServices/Recipe/Rcp.mprecipexml
```
Element gRecipeXmlMpLink (Type=mprecipexml)
  mapp.Recipe.Xml:
    Auditing = MpAudit
  Alarms = MpAlarmX
    mapp.AlarmX.Core.Configuration:
      [0]:
        Message = {$MpRecipeXml/Alarms/SaveFailed}
      [1]:
        Message = {$MpRecipeXml/Alarms/SaveFailedPartial}
        Disable = TRUE
      [2]:
        Message = {$MpRecipeXml/Alarms/LoadFailed}
      [3]:
        Message = {$MpRecipeXml/Alarms/LoadFailedPartial}
        Disable = TRUE
Element gRecipeXmlPreviewMpLink (Type=mprecipexml)
  Alarms = MpAlarmX
    mapp.AlarmX.Core.Configuration:
      [0]:
        Message = {$MpRecipeXml/Alarms/SaveFailed}
        Severity = 10
      [1]:
        Message = {$MpRecipeXml/Alarms/SaveFailedPartial}
        Severity = 10
        Disable = TRUE
      [2]:
        Message = {$MpRecipeXml/Alarms/LoadFailed}
        Severity = 10
      [3]:
        Message = {$MpRecipeXml/Alarms/LoadFailedPartial}
        Severity = 10
        Disable = TRUE
```

### RecipeCSV.mprecipecsv - 5PPC2200_AL14_000/mappServices/Recipe/RecipeCSV.mprecipecsv
```
Element gRecipeCsvMpLink (Type=mprecipecsv)
  mapp.Recipe.Csv:
    Auditing = MpAudit
  Alarms = MpAlarmX
    mapp.AlarmX.Core.Configuration:
      [0]:
        Message = {$Recipe/Alarms/SaveFailed}
      [1]:
        Message = {$Recipe/Alarms/SaveFailedPartial}
      [2]:
        Message = {$Recipe/Alarms/LoadFailed}
      [3]:
        Message = {$Recipe/Alarms/LoadFailedPartial}
```

### RecipeFile.mpfilemanagerui - 5PPC2200_AL14_000/mappServices/Recipe/RecipeFile.mpfilemanagerui
```
Element gMpLinkFileManagerUIRecipe (Type=mpfilemanagerui)
  Alarms = MpAlarmX
```

### RecipeXML.mprecipexml - 5PPC2200_AL14_000/mappServices/Recipe/RecipeXML.mprecipexml
```
Element gRecipeXmlMpLink (Type=mprecipexml)
  mapp.Recipe.Xml:
    Auditing = MpAudit
  Alarms = MpAlarmX
    mapp.AlarmX.Core.Configuration:
      [0]:
        Message = {$Recipe/Alarms/SaveFailed}
      [1]:
        Message = {$Recipe/Alarms/SaveFailedPartial}
        Disable = TRUE
      [2]:
        Message = {$Recipe/Alarms/LoadFailed}
      [3]:
        Message = {$Recipe/Alarms/LoadFailedPartial}
        Disable = TRUE
```

### Report.mpreportcore - 5PPC2200_AL14_000/mappServices/Report/Report.mpreportcore
```
Element gMpLinkReport (Type=mpreportcore)
  MpReport:
    Settings:
      ResourceDeviceName = mappReport
      LanguageDependent:
        [0]:
          Language = en
          Font = 1
        [1]:
          Language = zh-CN
    PageLayouts:
      [0]:
        Name = Default
    Styles:
      Text:
        [0]:
          Name = Default
          Size = 12
        [1]:
          Name = Header
          Style = 1
          Size = 20
          Color = FF9900
        [2]:
          Name = Subheader
          Size = 16
          Color = FF9900
      Table:
        [0]:
          Name = Default
          Padding = 10
      Line:
        [0]:
          Name = Default
          Color = FF9900
      Chart:
        PieChart:
          [0]:
            Name = Default
            BorderWidth = 0
        LineChart:
          [0]:
            Name = Default
        BarChart:
          [0]:
            Name = Default
    Tables:
      [0]:
        Name = Information
        TableStyle = Default
        TextStyle = Default
        [0]:
          [0] = TextId
            Source = RecipeName
            Width = 50
          [1] = ValueId
            Value:
              ProcessVariable = ::RecipeMgt:MpRecipe_0.Info.LastLoadedRecipe
            Width = 50
        [1]:
          [0] = TextId
            Source = Index
            Width = 50
          [1] = TextId
            Source = Length [mm]
            Width = 50
          [2] = TextId
            Source = Number
            Width = 50
        [2]:
          [0] = TextId
            Source = 1
            Width = 50
          [1] = ValueId
            Value:
              ProcessVariable = ::MainCtrl:MainCtrl.Para.ProductLength[0]
            Width = 50
          [2] = ValueId
            Value:
              ProcessVariable = ::MainCtrl:MainCtrl.Para.ProductNumber[0]
            Width = 50
        [3]:
          [0] = TextId
            Source = 2
            Width = 50
          [1] = ValueId
            Value:
              ProcessVariable = ::MainCtrl:MainCtrl.Para.ProductLength[1]
            Width = 50
          [2] = ValueId
            Value:
              ProcessVariable = ::MainCtrl:MainCtrl.Para.ProductNumber[1]
            Width = 50
        [4]:
          [0] = TextId
            Source = 3
            Width = 50
          [1] = ValueId
            Value:
              ProcessVariable = ::MainCtrl:MainCtrl.Para.ProductLength[2]
            Width = 50
          [2] = ValueId
            Value:
              ProcessVariable = ::MainCtrl:MainCtrl.Para.ProductNumber[2]
            Width = 50
        [5]:
          [0] = TextId
            Source = 4
            Width = 50
          [1] = ValueId
            Value:
              ProcessVariable = ::MainCtrl:MainCtrl.Para.ProductLength[3]
            Width = 50
          [2] = ValueId
            Value:
              ProcessVariable = ::MainCtrl:MainCtrl.Para.ProductNumber[3]
            Width = 50
        [6]:
          [0] = TextId
            Source = 5
            Width = 50
          [1] = ValueId
            Value:
              ProcessVariable = ::MainCtrl:MainCtrl.Para.ProductLength[4]
            Width = 50
          [2] = ValueId
            Value:
              ProcessVariable = ::MainCtrl:MainCtrl.Para.ProductNumber[4]
            Width = 50
    Contents:
      [0]:
        Name = ContentHeader
        [0]:
          Text = {Header}
        [1] = DateTime
        [2] = Line
          LineStyle = Default
      [1]:
        Name = ContentTable
        [0] = Table
          Table = Information
          HorizontalAlign = 1
      [2]:
        Name = Header
        [0]:
          Text = Report of the Cross Cutter Machine
          HorizontalAlign = 1
          TextStyle = Header
      [3]:
        Name = EmptyLine
        [0] = EmptyLine
      [4]:
        Name = Underline
        [0] = Line
          LineStyle = Default
      [5]:
        Name = Date
        [0] = DateTime
          TextStyle = Default
    Reports:
      [0]:
        Name = Report
        PageLayout = Default
        Header = Header
        [0]:
          [0]:
            Content = Underline
        [1]:
          [0]:
            Content = EmptyLine
        [2]:
          Heading:
            Text = Time
            TextStyle = Subheader
          [0]:
            Content = Date
        [3]:
          [0]:
            Content = EmptyLine
        [4]:
          [0]:
            Content = EmptyLine
        [5]:
          Heading:
            Text = Data
            TextStyle = Subheader
          [0]:
            Content = ContentTable
  Alarms = MpAlarmX
    mapp.AlarmX.Core.Configuration:
      [0]:
        Message = {$Report/Alarms/GenerateFailed}
```

### ReportFile.mpfilemanagerui - 5PPC2200_AL14_000/mappServices/Report/ReportFile.mpfilemanagerui
```
Element gMpLinkFileManagerUIReport (Type=mpfilemanagerui)
  Alarms = MpAlarmX
    mapp.AlarmX.Core.Configuration:
      [0]:
        Message = {$File/Alarms/DeviceNotFound}
      [1]:
        Message = {$File/Alarms/AlreadyExisting}
      [2]:
        Message = {$File/Alarms/FileSystemError}
```

### UsX.mpuserx - 5PPC2200_AL14_000/mappServices/UserX/UsX.mpuserx
```
Element UserMgmtX (Type=mpuserx)
  Mgr:
    PasswordLength = 1
    LoginAttempts = 5
  ServerSettings:
    Server:
      AdditionalUserData:
        [0] = mail
        [1] = telephoneNumber
  Users:
    DefUser#1:
      id = Admin
      name = Admin
    DefUser#2:
      id = Anonymous
      name = Anonymous
    DefUser#3:
      id = Operator
      name = Operator
    DefUser#4:
      id = Service_Tech
      name = Service_Tech
  Groups:
    DefGroup#1:
      id = Administrators
      level = 100
      admin = TRUE
      rights:
        [0] = FullAccess
        [1] = ViewOnly
        [2] = StartOnly
    DefGroup#2:
      id = Everyone
      level = 3
      rights:
        [0] = ViewOnly
    DefGroup#3:
      id = Operators
      level = 30
      rights:
        [0] = StartOnly
    DefGroup#4:
      id = Service
      level = 50
      rights:
        [0] = StartOnly
        [1] = ViewOnly
```

### UserX.mpuserx - 5PPC2200_AL14_000/mappServices/UserX/UserX.mpuserx
```
Element UserMgmtX (Type=mpuserx)
  Mgr:
    PasswordChangeInterval = 7776000
    PasswordExpirationNotification = 864000
    UserExpirationTime = 31536000
    PasswordAlpha = TRUE
    PasswordLength = 6
    UserNameLength = 3
    LoginAttempts = 5
  ServerSettings:
    Server:
      AdditionalUserData:
        [0] = mail
        [1] = telephoneNumber
  Users:
    DefUser#1:
      id = Admin
      name = Admin
      lang = en
      unit = imperial
    DefUser#2:
      id = Anonymous
      name = Anonymous
      lang = en
      unit = metric
    DefUser#3:
      id = Operator
      name = Operator
      lang = en
      unit = imperial-us
    DefUser#4:
      id = Service_Tech
      name = Service_Tech
      lang = zh
      unit = metric
  Groups:
    DefGroup#1:
      id = Administrators
      level = 100
      admin = TRUE
      rights:
        [0] = FullAccess
        [1] = ViewOnly
        [2] = StartOnly
    DefGroup#2:
      id = Everyone
      level = 3
      rights:
        [0] = ViewOnly
    DefGroup#3:
      id = Operators
      level = 30
      rights:
        [0] = StartOnly
    DefGroup#4:
      id = Service
      level = 50
      rights:
        [0] = StartOnly
        [1] = ViewOnly
```

### UserXlogin.mpuserxlogin - 5PPC2200_AL14_000/mappServices/UserX/UserXlogin.mpuserxlogin
```
Element gMpLinkUserXLogin (Type=mpuserxlogin)
  Alarms = MpAlarmX
```

## Configuration TS_UnitTest_Sample

CPU , AutomationRuntime C4.91, Build 6.3.0, Safety 0.0

### Task classes (Cpu.sw)
```
Cyclic#1:
  AxisMgr <- MachineControl.AxisTemplate.AxisMgr.prg
  prototypeT <- MachineControl.AxisTemplate.UnitTests.prototypeTest.prg
Binaries: iomap, asfw, arconfig, ashwd, sysconf
Libraries: Runtime, sys_lib, AsIecCon, astime, AsARCfg, AsBrStr, UnitTest, LibAssert1, UtWs, UtMgr, SPLMyCalc, CoTrace, MpFile, MpData, MpBase, MpAxis, MpWebXs, MpAudit, MpRecipe, MpUserX, MpReport, MpTool, MpAlarmX, MpCom, MpBackup, McAxis, McBase, McAxGroup, McAcpAx, McPathGen, McPureVAx, McAcpPar, AsZip, FileIO, DataObj, brsystem, AsArSdm, MpServer, operator, standard, asstring, AsBrWStr, ArUser, AsMem, MTTypes, AsUPS, AsIO, AsIOMMan, Gat, IoMapMan, ArCfgMan, MTBasics, AsUSB, MpRegMark, dvframe
```

### Cutter.regmarkdetection - PC_any/mappControl/Cutter.regmarkdetection
```
Element gRegMarkDetection_Cutter (Type=regmarkdetection)
  RegistrationMarkDetection:
    SensorSignal:
      AxisReference = gAxisCrossCutter
      DelayCompensation:
        AdditionalDelayTime  // 0.
    Measurement = MarkToCylinder
      Product:
        Position:
          AxisReference = gAxisConveyor
          Source = SetValue
        Length:
          Value = 70
    Detection = MiddleOfEdges
      SetMarkPosition = 0
      ExpectationWindow:
        Width = 25
      MarkWidthMonitoring:
        MinimumWidth = 7
        MaximumWidth = 15
      MissedMarkReaction:
        MarkPosition = LastValue
        AutomaticSearch = Used
          AdditionalExpectationWindowShift = 25
    OutputSignals:
      ActualMarkPosition = ::CrossCutte:RegistrationControl.ActualMarkPosition
      MarkPositionError = ::CrossCutte:RegistrationControl.MarkPositionError
      ActualProductLength = ::CrossCutte:RegistrationControl.ActualProductLength
      ActualIntervalLength = ::CrossCutte:RegistrationControl.ActualIntervalLength
  Alarms = MpAlarmX
```

### AxTest.axis - PC_any/mappMotion/Prototype/AxTest.axis
```
Element gAxisTest (Type=axis)
  BaseTypeIsReadOnly = 0
  BaseType = LinearPeriodic
    MeasurementUnit = 5066068
    MeasurementResolutionIsReadOnly = 0
    MeasurementResolution = 0.01
    CountDirectionIsReadOnly = 0
    CountDirection = Standard
    PeriodSettings:
      Period = 70
  MovementLimitsIsReadOnly = 0
  MovementLimits = Internal
    Position:
      LowerLimitMin = -1.79769313486231E308
      UpperLimitMax = 1.79769313486231E308
      LowerLimit = -1000.0
      UpperLimit = 1000.0
    VelocityIsReadOnly = 0
    Velocity:
      VelocityMax = 3.4E38
      Velocity = 500
    AccelerationIsReadOnly = 0
    Acceleration:
      AccelerationMax = 3.4E38
      Acceleration = 5000
    DecelerationIsReadOnly = 0
    Deceleration:
      DecelerationMax = 3.4E38
      Deceleration = 50000
  Alarms = MpAlarmX
    mapp.AlarmX.Core.Configuration:
      [0]:
        Severity = 20
      [1]:
        Severity = 20
      [2]:
        Severity = 20
      [3]:
        Message = Operation problem {&Info} {&Name}
        Severity = 20
        AdditionalInformation1 = 
      [4]:
        Severity = 20
      [5]:
        Severity = 20
      [9]:
        Severity = 20
      [10]:
        Severity = 20
      [11]:
        Severity = 20
      [12]:
        Severity = 20
      [13]:
        Severity = 20
      [14]:
        Severity = 20
      [15]:
        Severity = 20
```

### VAxTest.purevaxcfg - PC_any/mappMotion/Prototype/VAxTest.purevaxcfg
```
Element PureVAxCfg_1 (Type=purevaxcfg)
  TypeID = PureVAxConfig
  PureVAxis:
    AxisReference = gAxisTest
    Homing:
      Mode = Direct
        Position = 0.0
        ReferencePulse = NotUsed
      RestorePositionVariable
    JerkFilter = NotUsed
```

### TestGrp.mpcomgroup - PC_any/mappServices/AxisTest/TestGrp.mpcomgroup
```
Element gGroupTest (Type=mpcomgroup)
  Linking:
    Subnodes:
      0 = gAxisTest
      1 = gAlarmXCore_Test
  Alarms = MpAlarmX
```

### MachineGrp.mpcomgroup - PC_any/mappServices/MachineGrp.mpcomgroup
```
Element gMpLinkGroup (Type=mpcomgroup)
  Linking:
    Subnodes:
      0 = gGroupTest
      1 = gMpLinkAlarmXCore
  Alarms = MpAlarmX
```

## Logical view

Binary libraries used (declarations not repeated): operator, runtime, astime, AsIecCon, brsystem, sys_lib, AsArSdm, FileIO, standard, AsBrStr, asstring, AsBrWStr, ArUser, AsMem, AsARCfg, MTTypes, AsZip, DataObj, AsUPS, AsIO, AsIOMMan, IoMapMan, ArCfgMan, MTBasics, AsUSB, CoTrace, MpBase, MpServer, MpRegMark, dvframe, McBase 5.16.2, MpAxis 5.16.2, McAcpAx 5.16.0, McPureVAx 5.16.0, McAxis 5.16.2, McAcpPar 5.16.0, MpWebXs 5.16.0, MpAudit 5.16.0, MpRecipe 5.16.1, MpUserX 5.16.0, MpReport 5.16.0, MpFile 5.16.0, MpData 5.16.0, MpAlarmX 5.16.0, MpCom 5.16.0, MpBackup 5.16.0, AsIODiag, McAxGroup 5.16.2, McPathGen 5.16.2, McProgInt 5.16.2, MpTool 5.16.2

### Global.typ - Global data types
```iecst
(*Visu-----------------------------------------------------*)

TYPE
	VisuCtl_typ : 	STRUCT  (*Structure Type for Visualization Control*)
		cmd : Visu_cmd_typ; (*Command of the Visualization *)
	END_STRUCT;
	Visu_cmd_typ : 	STRUCT  (*Structure Type for Visualization Commands*)
		bEnableArUser : BOOL; (*Diables/Enables The Display of User Management Page that usesAr User for User Management*)
		bEnableMpUserX : BOOL; (*Diables/Enables The Display of User Management Page that usesAr User for User Management*)
	END_STRUCT;
END_TYPE
```

### Global.var - Global variables
```iecst
(*Visualization Control Variable*)
VAR
	gSimulationActive : BOOL;
	gVisuCtrl : VisuCtl_typ; (*MyAxisParameters : MyAxisParametersType;*)
END_VAR
```

### Package Logical/Libraries - Global libraries

### Library Logical/Libraries/Gat (IEC)

#### GatDegreeToDistance.st
```iecst
(* This function translates a given degree and radius to the corresponding length on a linear axis
FUNCTION GatDegreeToDistance
	GatDegreeToDistance := (Degree / 360.0) * 2.0 * CONST_PI * Radius;
END_FUNCTION
```

#### GatIoForcingHandler.st
```iecst
(*********************************************************************************
 * Copyright: B&R Industrial Automation GmbH
 * Created:   27 July, 2021/16:41
 * Handles Io forcing
 *********************************************************************************)

(* Handles IO forcing for all modules *)
FUNCTION_BLOCK GatIoForcingHandler
	(* Function block not enabled *)
	IF NOT Enable THEN
		(* Close arcfg *)
		IF Internal.ArCfgIdent <> 0 THEN
			Internal.AR_CloseArCfg_Int.Ident := Internal.ArCfgIdent;
			Internal.AR_CloseArCfg_Int.Enable := TRUE;
			Internal.AR_CloseArCfg_Int.Store := FALSE;
			Internal.AR_CloseArCfg_Int();
			IF Internal.AR_CloseArCfg_Int.Status = ERR_OK THEN
				Internal.AR_CloseArCfg_Int.Enable := FALSE;
				Internal.AR_CloseArCfg_Int.Store := FALSE;
				Internal.AR_CloseArCfg_Int();
				Internal.ArCfgIdent := 0;
			END_IF
		END_IF
		(* Close iomap *)
		IF Internal.IoMapIdent <> 0 THEN
			Internal.IO_CloseIoMap_Int.Ident := Internal.IoMapIdent;
			Internal.IO_CloseIoMap_Int.Enable := TRUE;
			Internal.IO_CloseIoMap_Int.Store := FALSE;
			Internal.IO_CloseIoMap_Int();
			IF Internal.IO_CloseIoMap_Int.Status = ERR_OK THEN
				Internal.IO_CloseIoMap_Int.Enable := FALSE;
				Internal.IO_CloseIoMap_Int.Store := FALSE;
				Internal.IO_CloseIoMap_Int();
				Internal.IoMapIdent := 0;
			END_IF
		END_IF
		(* Function block disabled, return here *)
		Internal.InitState := 0;
		Internal.CommandState := 0;
		Internal.NrOfIoChannels := 0;
		Internal.NrOfModules := 0;
		Initializing := FALSE;
		Ready := FALSE;
		RETURN;
	END_IF

	(* Initialize Io module and channel structure *)
	IF NOT Ready THEN
		Initializing := TRUE;
		(* Open arcfg *)
		IF Internal.ArCfgIdent = 0 THEN
			Internal.InitState := 0;
			Internal.AR_OpenArCfg_Int.Enable := TRUE;
			Internal.AR_OpenArCfg_Int();
			IF Internal.AR_OpenArCfg_Int.Status = ERR_OK THEN
				Internal.ArCfgIdent := Internal.AR_OpenArCfg_Int.Ident;
				Internal.NrOfModules := AR_NumberOfModules(Internal.ArCfgIdent);
				Internal.AR_OpenArCfg_Int.Enable := FALSE;
				Internal.AR_OpenArCfg_Int();
			ELSE
				RETURN;
			END_IF
		END_IF
		(* Open iomap *)
		IF Internal.IoMapIdent = 0 THEN
			Internal.InitState := 0;
			Internal.IO_OpenIoMap_Int.Enable := TRUE;
			Internal.IO_OpenIoMap_Int();
			IF Internal.IO_OpenIoMap_Int.Status = ERR_OK THEN
				Internal.IdxIoChannel := 1;
				Internal.IoMapIdent := Internal.IO_OpenIoMap_Int.Ident;
				Internal.NrOfIoChannels := Internal.IO_OpenIoMap_Int.NumberOfChannels;
				Internal.IO_OpenIoMap_Int.Enable := FALSE;
				Internal.IO_OpenIoMap_Int();
				brsmemset(ADR(IoModules), 0, SIZEOF(IoModules));
			ELSE
				RETURN;
			END_IF
		END_IF

		(* iomap and arcfg are open, start initialization *)
		CASE Internal.InitState OF
			0: // Find all visible IoChannels and sort them by module path
				(* Loop through IoChannels *)
				IF IO_ReadChannel(Internal.IoMapIdent, Internal.IdxIoChannel, ADR(Internal.TempChannel.Type), ADR(Internal.TempChannel.Inverted),
					ADR(Internal.TempChannel.ChannelName), ADR(Internal.TempChannel.PvName), ADR(Internal.TempChannel.ModulePath), ADR(Internal.TempChannel.TaskClass)) THEN
					(* Check visibility *)
					IF (NOT GatIoIsVisible(ADR(Internal.TempChannel.ChannelName))) OR (brsstrlen(ADR(Internal.TempChannel.ModulePath)) = 0) THEN
						Internal.IdxIoChannel := Internal.IdxIoChannel + 1;
						IF Internal.IdxIoChannel > Internal.NrOfIoChannels THEN
							Internal.InitState := Internal.InitState + 1;
							Internal.IdxModule := 0;
						END_IF
						RETURN;
					END_IF
					(* Search related module *)
					FOR Internal.IdxModule := 0 TO gatMAX_IDX_IO_MODULES DO
						IF brsstrcmp(ADR(IoModules[Internal.IdxModule].ModulePath), ADR('')) = 0 THEN
							(* Related module not in list yet, add module *)
							brsstrcpy(ADR(IoModules[Internal.IdxModule].ModulePath), ADR(Internal.TempChannel.ModulePath));
						END_IF
						IF brsstrcmp(ADR(IoModules[Internal.IdxModule].ModulePath), ADR(Internal.TempChannel.ModulePath)) = 0 THEN
							(* Module found *)
							GatMakeIoDpName(Internal.TempChannel, ADR(Internal.TempChannel.IoForcing.DpName));
							IoModules[Internal.IdxModule].IoChannels[IoModules[Internal.IdxModule].NrOfIoChannels] := Internal.TempChannel;
							IoModules[Internal.IdxModule].NrOfIoChannels := IoModules[Internal.IdxModule].NrOfIoChannels + 1;
							Internal.IdxIoChannel := Internal.IdxIoChannel + 1;
							IF Internal.IdxIoChannel > Internal.NrOfIoChannels THEN
								Internal.InitState := Internal.InitState + 1;
								Internal.IdxModule := 0;
							END_IF
							RETURN;
						END_IF
					END_FOR
				END_IF

			1: // Add Module names to each io module
				(* Check if module index is populated *)
				IF brsstrlen(ADR(IoModules[Internal.IdxModule].ModulePath)) = 0 THEN
					Internal.IdxModule := Internal.IdxModule + 1;
					IF Internal.IdxModule > gatMAX_IDX_IO_MODULES THEN
						Internal.IdxModule := 0;
						Internal.IdxIoChannel := 0;
						Internal.InitState := Internal.InitState + 1;
					END_IF
					RETURN;
				END_IF
				(* Loop through modules in arcfg to find the correct name *)
				FOR Internal.IdxModuleNames := 1 TO Internal.NrOfModules DO
					AR_GetModuleInfo(Internal.ArCfgIdent, Internal.IdxModuleNames, ADR(IoModules[Internal.IdxModule].ModuleName), ADR(IoModules[Internal.IdxModule].ModulePath));
					IF brsstrcmp(ADR(IoModules[Internal.IdxModule].ModulePath), ADR(IoModules[Internal.IdxModule].IoChannels[0].ModulePath)) = 0 THEN
						(* Correct name was found *)
						Internal.IdxModule := Internal.IdxModule + 1;
						IF Internal.IdxModule > gatMAX_IDX_IO_MODULES THEN
							Internal.IdxModule := 0;
							Internal.IdxIoChannel := 0;
							Internal.InitState := Internal.InitState + 1;
						END_IF
						RETURN;
					END_IF
				END_FOR

			2: // Close iomap and arcfg
				Internal.AR_CloseArCfg_Int.Enable := TRUE;
				Internal.AR_CloseArCfg_Int.Ident := Internal.ArCfgIdent;
				Internal.AR_CloseArCfg_Int.Store := FALSE;
				Internal.IO_CloseIoMap_Int.Enable := TRUE;
				Internal.IO_CloseIoMap_Int.Ident := Internal.IoMapIdent;
				Internal.IO_CloseIoMap_Int.Store := FALSE;

				Internal.AR_CloseArCfg_Int();
				Internal.IO_CloseIoMap_Int();

				IF (Internal.AR_CloseArCfg_Int.Status = ERR_OK) AND (Internal.IO_CloseIoMap_Int.Status = ERR_OK) THEN
					Ready := TRUE;
					Initializing := FALSE;
					Internal.IoMapIdent := 0;
					Internal.ArCfgIdent := 0;
				END_IF
		END_CASE;
	ELSE // Ready = TRUE
		(* Check if current indices are populated *)
		WHILE (brsstrlen(ADR(IoModules[Internal.IdxModule].IoChannels[Internal.IdxIoChannel].ChannelName)) = 0)
			OR (SelectedRefreshMode AND NOT IoModules[Internal.IdxModule].IoChannels[Internal.IdxIoChannel].IoForcing.RefreshActualValue AND NOT (Internal.CommandState = 1)) DO
			Internal.IdxModule := Internal.IdxModule + 1;
			Internal.IdxIoChannel := 0;
			IF Internal.IdxModule > gatMAX_IDX_IO_MODULES THEN
				Internal.IdxModule := 0;
				RETURN;
			END_IF
		END_WHILE

		(* Set force value *)
		IF IoModules[Internal.IdxModule].IoChannels[Internal.IdxIoChannel].IoForcing.ForceValue <> Internal.ForceValue[Internal.IdxModule, Internal.IdxIoChannel] THEN
			Internal.AsIOSetForceValue_Int.enable := TRUE;
			Internal.AsIOSetForceValue_Int.pDatapoint := ADR(IoModules[Internal.IdxModule].IoChannels[Internal.IdxIoChannel].IoForcing.DpName);
			Internal.AsIOSetForceValue_Int.value := IoModules[Internal.IdxModule].IoChannels[Internal.IdxIoChannel].IoForcing.ForceValue;
			Internal.AsIOSetForceValue_Int();
			IF Internal.AsIOSetForceValue_Int.status = ERR_OK THEN
				Internal.AsIOSetForceValue_Int.enable := FALSE;
				Internal.AsIOSetForceValue_Int();
				Internal.ForceValue[Internal.IdxModule, Internal.IdxIoChannel] := IoModules[Internal.IdxModule].IoChannels[Internal.IdxIoChannel].IoForcing.ForceValue;
			END_IF
		END_IF
		(* Enable/Disable forcing *)
		IF IoModules[Internal.IdxModule].IoChannels[Internal.IdxIoChannel].IoForcing.SetForceActive <> Internal.ForceEnabled[Internal.IdxModule, Internal.IdxIoChannel] THEN
			IF IoModules[Internal.IdxModule].IoChannels[Internal.IdxIoChannel].IoForcing.SetForceActive THEN
				Internal.AsIOEnableForcing_Int.enable := TRUE;
				Internal.AsIOEnableForcing_Int.pDatapoint := ADR(IoModules[Internal.IdxModule].IoChannels[Internal.IdxIoChannel].IoForcing.DpName);
				Internal.AsIOEnableForcing_Int();
				IF (Internal.AsIOEnableForcing_Int.status = ERR_OK) THEN
					Internal.AsIOEnableForcing_Int.enable := FALSE;
					Internal.AsIOEnableForcing_Int();
					Internal.ForceEnabled[Internal.IdxModule, Internal.IdxIoChannel] := TRUE;
				END_IF
			ELSE
				Internal.AsIODisableForcing_Int.enable := TRUE;
				Internal.AsIODisableForcing_Int.pDatapoint := ADR(IoModules[Internal.IdxModule].IoChannels[Internal.IdxIoChannel].IoForcing.DpName);
				Internal.AsIODisableForcing_Int();
				IF (Internal.AsIODisableForcing_Int.status = ERR_OK) THEN
					Internal.AsIODisableForcing_Int.enable := FALSE;
					Internal.AsIODisableForcing_Int();
					Internal.ForceEnabled[Internal.IdxModule, Internal.IdxIoChannel] := FALSE;
				END_IF
			END_IF
		END_IF
		(* Set actual value *)
		Internal.AsIODPStatus_Int.enable := TRUE;
		Internal.AsIODPStatus_Int.pDatapoint := ADR(IoModules[Internal.IdxModule].IoChannels[Internal.IdxIoChannel].IoForcing.DpName);
		Internal.AsIODPStatus_Int();
		IF Internal.AsIODPStatus_Int.status = ERR_OK THEN
			IF Internal.AsIODPStatus_Int.flags.2 THEN
				IoModules[Internal.IdxModule].IoChannels[Internal.IdxIoChannel].IoForcing.ActualValue := Internal.AsIODPStatus_Int.forceValue;
			ELSE
				IoModules[Internal.IdxModule].IoChannels[Internal.IdxIoChannel].IoForcing.ActualValue := Internal.AsIODPStatus_Int.value;
			END_IF
			Internal.AsIODPStatus_Int.enable := FALSE;
			Internal.AsIODPStatus_Int();
		END_IF
		(* Go to next index when nothing to do *)
		IF ((Internal.AsIOSetForceValue_Int.status = ERR_FUB_ENABLE_FALSE) OR (Internal.AsIOSetForceValue_Int.status = ERR_OK))
			AND ((Internal.AsIOEnableForcing_Int.status = ERR_FUB_ENABLE_FALSE) OR (Internal.AsIOEnableForcing_Int.status = ERR_OK))
			AND ((Internal.AsIODisableForcing_Int.status = ERR_FUB_ENABLE_FALSE) OR (Internal.AsIODisableForcing_Int.status = ERR_OK))
			AND ((Internal.AsIODPStatus_Int.status = ERR_FUB_ENABLE_FALSE) OR (Internal.AsIODPStatus_Int.status = ERR_OK)) THEN
			Internal.IdxIoChannel := Internal.IdxIoChannel + 1;
			IF Internal.IdxIoChannel > gatMAX_IDX_IO_CHANNELS THEN
				Internal.IdxIoChannel := 0;
				Internal.IdxModule := Internal.IdxModule + 1;
			END_IF
			IF Internal.IdxModule > gatMAX_IDX_IO_MODULES THEN
				Internal.IdxModule := 0;
			END_IF
			(* Handle command inputs *)
			CASE Internal.CommandState OF
				0: (* Wait for command *)
					IF ResetAllForcing THEN
						FOR Internal.IdxModuleCmd := 0 TO gatMAX_IDX_IO_MODULES DO
							FOR Internal.IdxIoChannelCmd := 0 TO gatMAX_IDX_IO_CHANNELS DO
								IoModules[Internal.IdxModuleCmd].IoChannels[Internal.IdxIoChannelCmd].IoForcing.SetForceActive := FALSE;
							END_FOR
						END_FOR
						CommandBusy := TRUE;
						Internal.CommandState := 1;
					END_IF
				1: (* ResetAllForcing *)
					CommandBusy := TRUE;
					FOR Internal.IdxModuleCmd := 0 TO gatMAX_IDX_IO_MODULES DO
						FOR Internal.IdxIoChannelCmd := 0 TO gatMAX_IDX_IO_CHANNELS DO
							IF Internal.ForceEnabled[Internal.IdxModuleCmd, Internal.IdxIoChannelCmd] THEN
								RETURN;
							END_IF
						END_FOR
					END_FOR
					(* All forcing is disabled *)
					CommandBusy := FALSE;
					CommandDone := TRUE;
					Internal.CommandState := 10;
				10: (* Command done *)
					CommandDone := TRUE;
					IF NOT ResetAllForcing THEN
						CommandDone := FALSE;
						Internal.CommandState := 0;
					END_IF
			END_CASE;
		END_IF
	END_IF
END_FUNCTION_BLOCK

(* Creates the IO data point name from the given information *)
FUNCTION GatMakeIoDpName
	brsmemset(ADR(DpName), 0, SIZEOF(DpName));

	CASE IoChannel.Type OF
		IO_DIG_INPUT:
			brsstrcpy(ADR(DpName), ADR('%IX.'));

		IO_DIG_OUTPUT:
			brsstrcpy(ADR(DpName), ADR('%QX.'));

		IO_ANA_INPUT:
			brsstrcpy(ADR(DpName), ADR('%IW.'));

		IO_TEMP_INPUT:
			brsstrcpy(ADR(DpName), ADR('%IW.'));

		IO_RESISTOR_INPUT:
			brsstrcpy(ADR(DpName), ADR('%IW.'));

		IO_ANA_OUTPUT:
			brsstrcpy(ADR(DpName), ADR('%QW.'));

		IO_PWM_OUTPUT:
			brsstrcpy(ADR(DpName), ADR('%QW.'));

		IO_USINT_INPUT:
			brsstrcpy(ADR(DpName), ADR('%IB.'));

		IO_USINT_OUTPUT:
			brsstrcpy(ADR(DpName), ADR('%QB.'));

		IO_UDINT_INPUT:
			brsstrcpy(ADR(DpName), ADR('%ID.'));

		IO_UDINT_OUTPUT:
			brsstrcpy(ADR(DpName), ADR('%QD.'));
	END_CASE;

	brsstrcat(ADR(DpName), ADR(IoChannel.ModulePath));
	brsstrcat(ADR(DpName), ADR('.'));
	brsstrcat(ADR(DpName), ADR(IoChannel.ChannelName));

	GatMakeIoDpName := TRUE;
END_FUNCTION

(* Determines whether an IO channel should be accessible on the HMI *)
FUNCTION GatIoIsVisible
	GatIoIsVisible := TRUE;
	IF (brsmemcmp(ADR(ChannelName), ADR('DigitalOutput'), 13) = 0) THEN
		RETURN;
	END_IF
	IF (brsmemcmp(ADR(ChannelName), ADR('DigitalInput'), 12) = 0) THEN
		RETURN;
	END_IF
	IF (brsmemcmp(ADR(ChannelName), ADR('CounterInput'), 12) = 0) THEN
		RETURN;
	END_IF
	IF (brsmemcmp(ADR(ChannelName), ADR('AnalogOutput'), 12) = 0) THEN
		RETURN;
	END_IF
	IF (brsmemcmp(ADR(ChannelName), ADR('AnalogInput'), 11) = 0) THEN
		RETURN;
	END_IF
	IF (brsmemcmp(ADR(ChannelName), ADR('Temperature'), 11) = 0) THEN
		RETURN;
	END_IF
	IF (brsmemcmp(ADR(ChannelName), ADR('RelayOutput'), 11) = 0) THEN
		RETURN;
	END_IF
	IF (brsmemcmp(ADR(ChannelName), ADR('PulseWidthCurrentPwm'), 20) = 0) THEN
		RETURN;
	END_IF
	IF (brsmemcmp(ADR(ChannelName), ADR('PulseWidthCurrentPWM'), 20) = 0) THEN
		RETURN;
	END_IF
	IF (brsmemcmp(ADR(ChannelName), ADR('Counter'), 7) = 0) THEN
		RETURN;
	END_IF
	GatIoIsVisible := FALSE;
	RETURN;
END_FUNCTION
```

### Package Logical/Infrastructure - Package for Machine Infrastructure

### mappFrameworkGlobal.var - Global variables for the mapp Framework
```iecst
VAR CONSTANT
	PARAMETERS_CATEGORY : STRING[10] := 'Parameters';
	MACHINE_CONFIGURATION_CATEGORY : STRING[30] := 'Machine Configuration';
	MAX_IDX_USB_DEV_LIST : USINT := 1; (*Max index for usb storage devices (1 means up to two devices with index 0 and 1)*)
END_VAR
VAR
	gUSBAvailable : ARRAY[0..MAX_IDX_USB_DEV_LIST] OF BOOL; (*Status array of USB storage devices*)
END_VAR
```

- Project.language - Project Language file (not shown)

### Package Logical/Infrastructure/AlarmX - Package for mapp AlarmX Framework

### Program Logical/Infrastructure/AlarmX/AlarmMgr (IEC) - Alarm manager

#### AlarmMgr.st
```iecst
//***********************************************************************
// Copyright: B&R Industrial Automation GmbH
// Author: B&R Industrial Automation GmbH
// Created: April 12, 2022
// Description: Tasks for alarm management.
//***********************************************************************

PROGRAM _INIT

	// Create folder for this component on the user file device
	DirCreate_0(enable := TRUE, pDevice := ADR('UserPartition'), pName := ADR(LOCAL_FOLDER));

	// Check if folder already exist and if so disabled the function block call
	IF DirCreate_0.status = fiERR_DIR_ALREADY_EXIST THEN
		DirCreate_0(enable := FALSE);
	END_IF

	// Call action to intialize alarm samples
	AlarmSampleInit;

	// Initialize mapp function blocks
	MpAlarmXCore_0.Enable := TRUE;
	MpAlarmXCore_0.MpLink := ADR(gMpLinkAlarmXCore);
	MpAlarmXCore_0();

	MpAlarmXHistory_0.Enable := TRUE;
	MpAlarmXHistory_0.DeviceName := ADR('mappAlarmXFiles');
	MpAlarmXHistory_0.MpLink := ADR(gMpLinkAlarmXHistory);
	MpAlarmXHistory_0();

	MpAlarmXListUI_0.Enable := TRUE;
	MpAlarmXListUI_0.UISetup.AlarmListScrollWindow := 10;
	MpAlarmXListUI_0.UISetup.AlarmListSize := 50;
	MpAlarmXListUI_0.UISetup.TimeStampPattern := '%Y %m %d %H:%M:%S';
	MpAlarmXListUI_0();

	MpAlarmXHistoryUI_0.Enable := TRUE;
	MpAlarmXHistoryUI_0.UISetup.AlarmListScrollWindow := 10;
	MpAlarmXHistoryUI_0.UISetup.AlarmListSize := (SIZEOF(MpAlarmXListUIConnect.AlarmList.InstanceID) / SIZEOF(MpAlarmXListUIConnect.AlarmList.InstanceID[0]));
	MpAlarmXHistoryUI_0.UISetup.TimeStampPattern := '%Y %m %d %H:%M:%S';
	MpAlarmXHistoryUI_0();

END_PROGRAM

PROGRAM _CYCLIC

	IF EDGEPOS(SafetyInputs.AcknowledgeAlarms) THEN
        MpAlarmXListUIConnect.AcknowledgeAll := TRUE;
	END_IF

	IF (HmiAlarmX.Commands.ExportAlarms = TRUE) THEN
		MpAlarmXHistory_0.Export := TRUE;
	END_IF

    // Call all cyclic actions
    AlarmHandling;
    GetBacktraceInformation;
    ExecuteQuery;
    QueryTableConfig;
    AlarmSampleFub;

	// Check if any reactions are active.
	// Typically the MpAlarmXCheckReaction() function is called from other tasks within the application.
	// For example, the axis control task might check for the 'Error' reaction to determine whether to send a stop command to the axes.
	// Therefore, copy/paste these IF statements to other places in the application as needed.
    IF MpAlarmXCheckReaction(gMpLinkAlarmXCore, 'Error') THEN
        // Error is active. Add code here to respond to error situation.
    ELSIF MpAlarmXCheckReaction(gMpLinkAlarmXCore, 'Warning') THEN
        // Warning is active. Add code here to respond to warning situation.
	ELSIF MpAlarmXCheckReaction(gMpLinkAlarmXCore, 'Info') THEN
        // Info is active. Add code here to resond to info situation.
	END_IF

	IF ((MpAlarmXHistory_0.Export = TRUE) AND (MpAlarmXHistory_0.CommandDone = TRUE)) THEN
		HmiAlarmX.Commands.ExportAlarms := FALSE;
		MpAlarmXHistory_0.Export := FALSE;
	END_IF

    // Error reset
    IF NOT MpAlarmXCore_0.Error THEN
        MpAlarmXCore_0.ErrorReset := FALSE;
    END_IF
    IF NOT MpAlarmXListUI_0.Error THEN
        MpAlarmXListUI_0.ErrorReset := FALSE;
    END_IF
    IF NOT MpAlarmXHistory_0.Error THEN
        MpAlarmXHistory_0.ErrorReset := FALSE;
    END_IF
    IF NOT MpAlarmXHistoryUI_0.Error THEN
        MpAlarmXHistoryUI_0.ErrorReset := FALSE;
    END_IF

	// Assign MpLinks & UIConnects
	MpAlarmXCore_0.MpLink := ADR(gMpLinkAlarmXCore);
	MpAlarmXListUI_0.MpLink := ADR(gMpLinkAlarmXCore);
	MpAlarmXListUI_0.UIConnect := ADR(MpAlarmXListUIConnect);
	MpAlarmXHistory_0.MpLink := ADR(gMpLinkAlarmXHistory);
	MpAlarmXHistoryUI_0.MpLink := ADR(gMpLinkAlarmXHistory);
	MpAlarmXHistoryUI_0.UIConnect := ADR(MpAlarmXHistoryUIConnect);

	// Call function blocks
	MpAlarmXCore_0();
	MpAlarmXListUI_0();
	MpAlarmXHistory_0();
	MpAlarmXHistoryUI_0();

END_PROGRAM

PROGRAM _EXIT

	// Disable the function blocls to unlink the MpLinks
    MpAlarmXCore_0.Enable := FALSE;
    MpAlarmXListUI_0.Enable := FALSE;
    MpAlarmXHistory_0.Enable := FALSE;
	MpAlarmXHistoryUI_0.Enable := FALSE;
	QueryActiveAlarms_0.Enable := FALSE;

	// Call function blocks
    MpAlarmXCore_0();
    MpAlarmXListUI_0();
    MpAlarmXHistory_0();
    MpAlarmXHistoryUI_0();
    QueryActiveAlarms_0();

END_PROGRAM
```

#### AlarmMgr.typ
```iecst
(*Structure types*)

TYPE
	AlarmHmiInterfaceType : 	STRUCT  (*Structure to hold commands and status from the HMI*)
		Commands : AlarmCommandsType; (*HMI commands*)
		Status : {REDUND_UNREPLICABLE} AlarmStatusType; (*HMI status*)
	END_STRUCT;
	AlarmCommandsType : 	STRUCT  (*Structure to hold the commands from the HMI*)
		ExportAlarms : BOOL; (*Triggers an alarm export of the alarm history. Connected to a button on the HMI. *)
		RunQuery : BOOL; (*Triggers the query to run. Connected to a button on the HMI. *)
	END_STRUCT;
	AlarmStatusType : 	STRUCT  (*Structure to hold status information from the mapp View HMI. (This structure is not compatible/relevant if you are using a VC4 visualization)*)
		AlarmHistSortCfg : STRING[1000]; (*Sort configuration property for the AlarmHistory widget *)
		AlarmHistFilterCfg : STRING[1000]; (*Filter configuration property for the AlarmHistory widget*)
		AlarmSortCfg : STRING[1000]; (*Sort configuration for the AlarmList widget*)
		AlarmFilterCfg : STRING[1000]; (*Filter configuration for the AlarmList widget*)
		TableConfig : ARRAY[0..1]OF STRING[120]; (*Table configuration for the alarm query Table*)
		Query : AlarmQueryHMIType; (*Structure which rearranges the query data from AlarmQuery into a structure of arrays for easy connection to the Table widget*)
		InstanceID : UINT; (*The instanceID of the alarm that was most recently clicked in the AlarmList. Set by an eventbinding in mapp View*)
	END_STRUCT;
	AlarmQueryType : 	STRUCT  (*Structure for query results and status*)
		State : ActiveAlarmStateEnum; (*State variable for the query state machine*)
		LastUpdateCount : UDINT; (*Previous count of query results. Used to check for new query data. *)
		UpdateCount : UDINT; (*Count of query results. Increases each time new results are availble. *)
		Alarms : ARRAY[0..MAX_QUERY_RESULTS]OF AlarmType; (*Query data*)
		Next : BOOL; (*Trigger to query the next data, if there are more results than MAX_QUERY_RESULTS*)
	END_STRUCT;
	AlarmQueryHMIType : 	STRUCT  (*Datatype for the structure which rearranges the query data from AlarmQuery into a structure of arrays for easy connection to the Table widget in mapp View*)
		Active : ARRAY[0..MAX_QUERY_RESULTS]OF BOOL; (*StateActive array*)
		Acknowledged : ARRAY[0..MAX_QUERY_RESULTS]OF BOOL; (*StateAcknowledged array*)
		Scope : ARRAY[0..MAX_QUERY_RESULTS]OF WSTRING[80]; (*Scope array*)
		Name : ARRAY[0..MAX_QUERY_RESULTS]OF STRING[80]; (*Name array*)
		Message : ARRAY[0..MAX_QUERY_RESULTS]OF WSTRING[255]; (*Message array*)
		AdditionalInfo : ARRAY[0..MAX_QUERY_RESULTS]OF WSTRING[255]; (*AdditionalInformation1 array*)
		TimeStamp : ARRAY[0..MAX_QUERY_RESULTS]OF DATE_AND_TIME; (*TimeStamp array*)
		Code : ARRAY[0..MAX_QUERY_RESULTS]OF UDINT; (*Code array*)
		Severity : ARRAY[0..MAX_QUERY_RESULTS]OF UDINT; (*Severity array*)
		QueryCount : USINT; (*Count of query results for building the query table configuration string*)
	END_STRUCT;
	AlarmType : 	STRUCT  (*Structure to hold the alarm data for the query results*)
		Active : BOOL; (*ActiveAlarms query, StateActive column*)
		Acknowledged : BOOL; (*ActiveAlarms query, StateAcknowledged column*)
		Scope : WSTRING[80]; (*ActiveAlarms query, Scope column*)
		Name : STRING[80]; (*ActiveAlarms query, Name column*)
		Message : WSTRING[255]; (*ActiveAlarms query, Message column*)
		AdditionalInfo : WSTRING[255]; (*ActiveAlarms query, AdditionalInformation1*)
		TimeStamp : DATE_AND_TIME; (*ActiveAlarms query, TimeStamp column*)
		Code : UDINT; (*ActiveAlarms query, Code column*)
		Severity : UDINT; (*ActiveAlarms query, Severity column*)
	END_STRUCT;
	MachineDigitalInputsType : 	STRUCT  (*Safety related digital inputs *)
		EmergencyStop : ARRAY[0..MAX_ESTOP]OF BOOL; (*Emergency stop input signals*)
		SafetyDoor : ARRAY[0..MAX_SAFETY_DOOR]OF BOOL; (*Safety door input signals*)
		AcknowledgeAlarms : BOOL; (*Reset button input signal*)
	END_STRUCT;
	AlarmExamplesType : 	STRUCT  (*Structure for alarm samples*)
		LevelMonitoring : INT; (*Triggers LevelMonitoringExample alarm depending on the value set (<20 or >80)*)
		DeviationMonitoring : INT; (*Triggers the DeviationMonitoringExample alarm if this differs from DevationMonitoringSetpoint (below) by more than 5 units*)
		DeviationMonitoringSetpoint : INT; (*Setpoint for the DeviationMonitoringExample alarm. If DeviationMonitoring (above) differs from this value by more than 5 units, the alarm triggers*)
		RateOfChange : INT; (*Triggers the RateOfChangeExample alarm if this value changes at a rate of more than 5 units per second*)
		SnippetValue : INT; (*Process variable used in the SnippetExample alarm for the snippet*)
		SetControlExample : BOOL; (*Boolean to trigger the example alarm which is triggerd by MpAlarmXControlExample_0*)
	END_STRUCT;
END_TYPE

(*Enumerations*)

TYPE
	ActiveAlarmStateEnum :
		( (*Enumeration for the state for the query state machine*)
		ACTIVE_ALARM_WAIT, (*Wait state*)
		ACTIVE_ALARM_QUERY, (*State to query the alarm data*)
		ACTIVE_ALARM_NEXT (*State to check if more alarms meet the query criteria and need to be queried*)
		);
END_TYPE
```

#### AlarmMgr.var - Local variables
```iecst
(*Function Blocks*)
VAR
	HmiAlarmX : AlarmHmiInterfaceType; (*HMI interface structure*)
	MpAlarmXHistory_0 : MpAlarmXHistory; (*MpAlarmXHistory instance*)
	MpAlarmXHistoryUI_0 : MpAlarmXHistoryUI; (*MpAlarmXHistoryUI instance*)
	MpAlarmXListUI_0 : MpAlarmXListUI; (*MpAlarmXList instance*)
	MpAlarmXCore_0 : MpAlarmXCore; (*MpAlarmXCore instance*) (*ChangeStyleAlarmButton : USINT := 0; (*changeStyle of a AlarmFlyout in mappView*)
	MpAlarmXControlExample_0 : {REDUND_UNREPLICABLE} MpAlarmXAlarmControl; (*MpAlarmXAlarmControl instance*)
	QueryActiveAlarms_0 : {REDUND_UNREPLICABLE} MpAlarmXQuery; (*MpAlarmXQuery instance*)
	DirCreate_0 : DirCreate; (*DirCreate instance*)
END_VAR
(*Constants*)
VAR CONSTANT
	MAX_QUERY_RESULTS : USINT := 19; (*Maximum number of query results (Value+1)*)
	MAX_SAFETY_DOOR : UINT := 5; (*Maximum number of safety doors (Value+1)*)
	MAX_ESTOP : UINT := 2; (*Maximum number of emergency stops (Value+1)*)
	LOCAL_FOLDER : STRING[10] := 'AlarmX'; (*Folder name on the file device for AlarmX files*)
END_VAR
(*Structure Types*)
VAR
	MpAlarmXListUIConnect : MpAlarmXListUIConnectType := (0); (*AlarmX list connection to the UI*)
	MpAlarmXHistoryUIConnect : MpAlarmXHistoryUIConnectType; (*AlarmX History connection to the UI*)
	SafetyInputs : MachineDigitalInputsType; (*Safety related digital inputs*)
	AlarmExamples : {REDUND_UNREPLICABLE} AlarmExamplesType; (*Sample alarms for different monitoring types*)
	AlarmQuery : {REDUND_UNREPLICABLE} AlarmQueryType; (*Query results and status*)
END_VAR
(*Variables*)
VAR
	Alarms : {REDUND_UNREPLICABLE} ARRAY[0..99] OF BOOL; (*Array of monitored alarm bits*)
	CommissioningModeActive : {REDUND_UNREPLICABLE} BOOL; (*Boolean value to enable commissioning mode. By default, this inhibits the Alarms[0] alarm*)
	i : USINT; (*Index for loops*)
	MaxIndex : USINT; (*Maximum index for the alarm list*)
END_VAR
```

#### HMIActions.st
```iecst
ACTION GetBacktraceInformation:

    MaxIndex := (SIZEOF(MpAlarmXListUIConnect.AlarmList.InstanceID)/SIZEOF(MpAlarmXListUIConnect.AlarmList.InstanceID[0])) - 1;
    // Find selected alarm in order to show backtrace information
    FOR i := 0 TO MaxIndex DO
        IF (MpAlarmXCore_0.PendingAlarms = 0) THEN
            // No pending alarms, reset instance id
			HmiAlarmX.Status.InstanceID := 0;
			EXIT;
        END_IF

        IF (MpAlarmXListUIConnect.AlarmList.InstanceID[i] = HmiAlarmX.Status.InstanceID) THEN
            // Found an alarm
            MpAlarmXListUIConnect.AlarmList.SelectedIndex := i;
            EXIT;
        END_IF

        IF (MpAlarmXListUIConnect.AlarmList.InstanceID[i] = 0) THEN
            IF (MpAlarmXCore_0.PendingAlarms > i) THEN
                // Alarm not found, list can page up
                MpAlarmXListUIConnect.AlarmList.PageUp := TRUE;
            END_IF
			EXIT;
        ELSIF (i = MaxIndex) THEN
            // Alarm not found, list can page down
            MpAlarmXListUIConnect.AlarmList.PageDown := TRUE;
        END_IF
	END_FOR

END_ACTION

ACTION QueryTableConfig:

	// Configure visible list
	HmiAlarmX.Status.TableConfig[0] := '{ "specRows": [{"from":';
    FOR i := 0 TO 9 DO
        IF HmiAlarmX.Status.Query.Message[i] <> "" THEN
			HmiAlarmX.Status.Query.QueryCount := i + 1;
		END_IF
    END_FOR
    brsitoa((HmiAlarmX.Status.Query.QueryCount), ADR(HmiAlarmX.Status.TableConfig[0]) + brsstrlen(ADR(HmiAlarmX.Status.TableConfig[0])));
    brsstrcat(ADR(HmiAlarmX.Status.TableConfig[0]),  ADR(',"to":19, "visible":false}]}'));

END_ACTION
```

#### ExecuteQuery.st
```iecst
ACTION ExecuteQuery:

	// Initialize mapp function block
	QueryActiveAlarms_0.MpLink := ADR(gMpLinkAlarmXCore);
	QueryActiveAlarms_0.Enable := TRUE;
	QueryActiveAlarms_0.Name := ADR('ActiveAlarms');
	QueryActiveAlarms_0.Language := ADR('en');
	QueryActiveAlarms_0();

	CASE (AlarmQuery.State) OF
		ACTIVE_ALARM_WAIT:
			// Wait until the RunQuery command is triggered from the HMI.
			// If you prefer that the query runs anytime new data is available, then uncomment line 15 and comment out line 16 and delete
			// the "Run query" button from the HMI.
//			IF (AlarmQuery.LastUpdateCount <> AlarmQuery.UpdateCount) THEN
			IF (HmiAlarmX.Commands.RunQuery = TRUE) THEN
				brsmemset(ADR(AlarmQuery.Alarms[0]), 0, SIZEOF(AlarmQuery.Alarms));
				AlarmQuery.LastUpdateCount := AlarmQuery.UpdateCount;
				QueryActiveAlarms_0.Execute := TRUE;
				HmiAlarmX.Commands.RunQuery := FALSE;
				AlarmQuery.State := ACTIVE_ALARM_QUERY;
			END_IF

		ACTIVE_ALARM_QUERY:
			// If the number of query results is less than MAX_QUERY_RESULTS, return to the wait state
			IF ((QueryActiveAlarms_0.CommandDone = TRUE) AND (QueryActiveAlarms_0.Info.HasMoreRows = FALSE)) THEN
				QueryActiveAlarms_0.Execute := FALSE;
				QueryActiveAlarms_0.Next := FALSE;
				AlarmQuery.State := ACTIVE_ALARM_WAIT;
				// If the number of query results is more than MAX_QUERY_RESULTS, then query the next set of results
			ELSIF ((QueryActiveAlarms_0.CommandDone = TRUE) AND (QueryActiveAlarms_0.Info.HasMoreRows = TRUE)) THEN
				QueryActiveAlarms_0.Next := FALSE;
				AlarmQuery.State := ACTIVE_ALARM_NEXT;
			END_IF

		ACTIVE_ALARM_NEXT:
			IF (AlarmQuery.Next = TRUE) THEN
				// By default, AlarmQuery.Alarms has 20 elements, so it can hold 20 query results at a time (MAX_QUERY_RESULTS = 19).
				// If AlarmQuery.Next is true, this means the query result is more than 20 alarms.
				// If you want to save the data for the first 20 alarms, add code here to copy AlarmQuery.Alarms to another location.
				// Otherwise, the older alarms in the query will get overwritten with the newest entries here.
				brsmemset(ADR(AlarmQuery.Alarms[0]), 0, SIZEOF(AlarmQuery.Alarms));
				AlarmQuery.Next := FALSE;
				QueryActiveAlarms_0.Next := TRUE;
				AlarmQuery.State := ACTIVE_ALARM_QUERY;
			END_IF
	END_CASE

	// Convert the query results into arrays that can easily be bound to the Table widget in mapp View
	FOR i := 0 TO MAX_QUERY_RESULTS DO
		HmiAlarmX.Status.Query.Active[i] := AlarmQuery.Alarms[i].Active;
		HmiAlarmX.Status.Query.Acknowledged[i] := AlarmQuery.Alarms[i].Acknowledged;
		HmiAlarmX.Status.Query.Scope[i] := AlarmQuery.Alarms[i].Scope;
		HmiAlarmX.Status.Query.Name[i] := AlarmQuery.Alarms[i].Name;
		HmiAlarmX.Status.Query.Message[i] := AlarmQuery.Alarms[i].Message;
		HmiAlarmX.Status.Query.AdditionalInfo[i] := AlarmQuery.Alarms[i].AdditionalInfo;
		HmiAlarmX.Status.Query.TimeStamp[i] := AlarmQuery.Alarms[i].TimeStamp;
		HmiAlarmX.Status.Query.Severity[i] := AlarmQuery.Alarms[i].Severity;
	END_FOR

END_ACTION
```

#### AlarmSamples.st
```iecst
ACTION AlarmSampleInit:

    // Call all variables that are needed for the alarm examples and explain all examples in comments

    // If AlarmExamples.LevelMonitoring gets less than 20 or more than 80, the LevelMonitoringExample alarm will trigger
	// The Low limit is 20. The LowLow limit is 10. The High limit is 80. The HighHigh limit is 90.
    AlarmExamples.LevelMonitoring := 50;

	// If AlarmExamples.DeviationMonitoring deviates from the setpoint (AlarmExamples.DeviationMonitoringSetpoint) by more than 5
	// units in either direction, the DeviationMonitoringExample alarm will trigger
	AlarmExamples.DeviationMonitoring := 15;
	AlarmExamples.DeviationMonitoringSetpoint := 15;

	// If AlarmExamples.RateOfChange increases at a rate of more than 5 units per second, the RateOfChangeExample alarm will trigger
	AlarmExamples.RateOfChange := 0;

	// If AlarmExamples.SnippetValue gets between 50 and 100, an alarm will trigger and the current value will be shown in the alarm text
	AlarmExamples.SnippetValue := 10;

END_ACTION

ACTION AlarmSampleFub:

	// Example of using the MpAlarmXControl() function block.
	// Typically this function is called from other tasks within the application (decentralized).
	// For example, if you have an error in the recipe system, you can trigger it directly in the recipe task.
	// Therefore, copy/paste this example to other places in the application as needed.
    MpAlarmXControlExample_0.MpLink := ADR(gMpLinkAlarmXCore);
    MpAlarmXControlExample_0.Enable := TRUE;
    MpAlarmXControlExample_0.Name := ADR('MpAlarmXControlExample');
    MpAlarmXControlExample_0.Set := AlarmExamples.SetControlExample;
    MpAlarmXControlExample_0();

END_ACTION
```

#### AlarmMgt.typ - not listed in the package file held
```iecst
TYPE
	MachineDigitalInputsType : 	STRUCT  (*Safety related digital inputs of the machine*)
		EmergencyStop : ARRAY[0..MAX_IDX_ESTOP]OF BOOL; (*Emergency stop signal*)
		SafetyDoor : ARRAY[0..MAX_IDX_SAFETY_DOOR]OF BOOL; (*Safety door signal*)
		AcknowledgeAlarms : BOOL;
	END_STRUCT;
	AlarmExamplesType : 	STRUCT
		LevelMonitoring : INT;
		DeviationMonitoring : INT;
		DeviationMonitoringSetpoint : INT;
		RateOfChange : INT;
		SnippetValue : INT;
		SetControlExample : BOOL;
	END_STRUCT;
	ActiveAlarmStateEnum :
		(
		ACTIVE_ALARM_WAIT,
		ACTIVE_ALARM_QUERY,
		ACTIVE_ALARM_NEXT
		);
	AlarmType : 	STRUCT
		Active : BOOL;
		Acknowledged : BOOL;
		Scope : WSTRING[80];
		Name : STRING[80];
		Message : WSTRING[255];
		AdditionalInfo : WSTRING[255];
		TimeStamp : DATE_AND_TIME;
		Code : UDINT;
		Severity : UDINT;
	END_STRUCT;
	AlarmQueryType : 	STRUCT
		Next : BOOL;
		State : ActiveAlarmStateEnum;
		LastActiveAlarmUpdateCount : UDINT;
		ActiveAlarmUpdateCount : UDINT;
		Alarms : ARRAY[0..MAX_QUERY_RESULTS]OF AlarmType;
	END_STRUCT;
	AlarmHmiInterfaceType : 	STRUCT
		Commands : AlarmCommandsType;
		Status : {REDUND_UNREPLICABLE} AlarmStatusType;
	END_STRUCT;
	AlarmStatusType : 	STRUCT
		AlarmHistSortCfg : STRING[1000];
		AlarmHistFilterCfg : STRING[1000];
		AlarmSortCfg : STRING[1000];
		AlarmFilterCfg : STRING[1000];
		TableConfig : ARRAY[0..1]OF STRING[120];
	END_STRUCT;
	AlarmCommandsType : 	STRUCT
		ExportAlarms : BOOL;
		RunQuery : BOOL;
	END_STRUCT;
	AlarmQueryHMIType : 	STRUCT
		Active : ARRAY[0..MAX_QUERY_RESULTS]OF BOOL;
		Acknowledged : ARRAY[0..MAX_QUERY_RESULTS]OF BOOL;
		Scope : ARRAY[0..MAX_QUERY_RESULTS]OF WSTRING[80];
		Name : ARRAY[0..MAX_QUERY_RESULTS]OF STRING[80];
		Message : ARRAY[0..MAX_QUERY_RESULTS]OF WSTRING[255];
		AdditionalInfo : ARRAY[0..MAX_QUERY_RESULTS]OF WSTRING[255];
		TimeStamp : ARRAY[0..MAX_QUERY_RESULTS]OF DATE_AND_TIME;
		Code : ARRAY[0..MAX_QUERY_RESULTS]OF UDINT;
		Severity : ARRAY[0..MAX_QUERY_RESULTS]OF UDINT;
	END_STRUCT;
END_TYPE
```

#### AlarmMgt.var - not listed in the package file held
```iecst
(********************************************************************
 * COPYRIGHT -- Bernecker + Rainer
 ********************************************************************
 * Program: FolderHandling
 * File: FolderHandling.var
 * Author: Bernecker + Rainer
 * Created: December , 2020
 ********************************************************************
 * Local variables of program AlarmManagement
 ********************************************************************)
(*Function Blocks*)
VAR
	HmiAlarmX : AlarmHmiInterfaceType;
	MpAlarmXHistory_0 : MpAlarmXHistory; (*MpAlarmXHistory instance*)
	MpAlarmXHistoryUI_0 : MpAlarmXHistoryUI; (*MpAlarmXHistoryUI instance*)
	MpAlarmXListUI_0 : MpAlarmXListUI; (*MpAlarmXList instance*)
	MpAlarmXCore_0 : MpAlarmXCore; (*MpAlarmXCore instance*) (*ChangeStyleAlarmButton : USINT := 0; (*changeStyle of a AlarmFlyout in mappView*)
	DirCreate_New : DirCreate;
END_VAR
(*Alarm Management Variables*)
VAR
	Index : USINT; (*Index to loop through alarm list*)
	MaxIndex : USINT; (*Maximum index for the alarm list*)
	InstanceID : UINT; (*Instance ID*)
	MpAlarmXListUIConnect : MpAlarmXListUIConnectType := (0); (*AlarmVideo : WSTRING[255] := "";
	AlarmInfo : BOOL := 0;*)
	MpAlarmXHistoryUIConnect : MpAlarmXHistoryUIConnectType; (*AlarmX History connection to UI*)
	AlarmQuery : {REDUND_UNREPLICABLE} AlarmQueryType; (*Query Results*)
	QueryActiveAlarms : {REDUND_UNREPLICABLE} MpAlarmXQuery; (*MpAlarmXQuery instance*)
END_VAR
(*Safety Inputs*)
VAR
	SafetyInputs : MachineDigitalInputsType;
END_VAR
(*Defines*)
VAR CONSTANT
	MAX_IDX_ESTOP : UINT := 2;
	MAX_IDX_SAFETY_DOOR : UINT := 5;
	LOCAL_FOLDER : STRING[10] := 'AlarmX';
END_VAR
(*Examples*)
VAR
	CommissioningModeActive : {REDUND_UNREPLICABLE} BOOL; (*Inhibits the Alarms[0] alarm*)
	Alarms : {REDUND_UNREPLICABLE} ARRAY[0..99] OF BOOL; (*Array of active alarm*)
	AlarmExamples : {REDUND_UNREPLICABLE} AlarmExamplesType; (*Sample alarms for different monitoring types*)
	MpAlarmXControlExampleFB : {REDUND_UNREPLICABLE} MpAlarmXAlarmControl; (*MpAlarmXAlarmControl instance*)
END_VAR
VAR CONSTANT
	MAX_QUERY_RESULTS : USINT := 19;
END_VAR
VAR
	AlarmQueryHMI : AlarmQueryHMIType;
	i : USINT;
	EntryCount : USINT;
END_VAR
```

#### AlarmMgt.st - not listed in the package file held
```iecst
//***********************************************************************
// Copyright: B&R Industrial Automation GmbH
// Author: B&R Industrial Automation GmbH
// Created: Jan 1, 2022
// Description: Tasks for alarm control. The Alarm Management handling is
// done in this task.
//***********************************************************************

PROGRAM _INIT

	// Create folder for this component on the user file device
	DirCreate_New(enable := TRUE, pDevice := ADR('userPartition'), pName := ADR(LOCAL_FOLDER));

	// Check if folder already exist and if so disabled the function block call
	IF DirCreate_New.status = fiERR_DIR_ALREADY_EXIST THEN
		DirCreate_New(enable := FALSE);
	END_IF

	// Initialize mapp function blocks
	MpAlarmXCore_0.Enable := TRUE;
	MpAlarmXCore_0.MpLink := ADR(gMpLinkAlarmXCore);
	MpAlarmXCore_0();

	MpAlarmXHistory_0.Enable := TRUE;
	MpAlarmXHistory_0.DeviceName := ADR('mappAlarmXFiles');
	MpAlarmXHistory_0.MpLink := ADR(gMpLinkAlarmXHistory);
	MpAlarmXHistory_0();

	MpAlarmXListUI_0.Enable := TRUE;
	MpAlarmXListUI_0.UISetup.AlarmListScrollWindow := 10;
	MpAlarmXListUI_0.UISetup.AlarmListSize := 50;
	MpAlarmXListUI_0.UISetup.TimeStampPattern := '%Y %m %d %H:%M:%S';
	MpAlarmXListUI_0();

	MpAlarmXHistoryUI_0.Enable := TRUE;
	MpAlarmXHistoryUI_0.UISetup.AlarmListScrollWindow := 10;
    MpAlarmXHistoryUI_0.UISetup.AlarmListSize := (SIZEOF(MpAlarmXListUIConnect.AlarmList.InstanceID) / SIZEOF(MpAlarmXListUIConnect.AlarmList.InstanceID[0]));
	MpAlarmXHistoryUI_0.UISetup.TimeStampPattern := '%Y %m %d %H:%M:%S';
	MpAlarmXHistoryUI_0();

	// Call action to intialize alarm samples
	AlarmSampleInit;

END_PROGRAM

PROGRAM _CYCLIC

	IF EDGEPOS(SafetyInputs.AcknowledgeAlarms) THEN
        MpAlarmXListUIConnect.AcknowledgeAll := TRUE;
	END_IF

	IF (HmiAlarmX.Commands.ExportAlarms = TRUE) THEN
		MpAlarmXHistory_0.Export := TRUE;
	END_IF

    // Call all cyclic actions
    AlarmHandling;
    GetBacktraceInformation;
    ExecuteQuery;
    QueryTableConfig;
    AlarmSampleFub;

	// Check if any reactions are active.
	// Typically the MpAlarmXCheckReaction() function is called from other tasks within the application.
	// For example, the axis control task might check for the 'Error' reaction to determine whether to send a stop command to the axes.
	// Therefore, copy/paste these IF statements to other places in the application as needed.
    IF MpAlarmXCheckReaction(gMpLinkAlarmXCore, 'Error') THEN
        // Error is active. Add code here to respond to error situation.
    ELSIF MpAlarmXCheckReaction(gMpLinkAlarmXCore, 'Warning') THEN
        // Warning is active. Add code here to respond to warning situation.
	ELSIF MpAlarmXCheckReaction(gMpLinkAlarmXCore, 'Info') THEN
        // Info is active. Add code here to resond to info situation.
	END_IF

	IF ((MpAlarmXHistory_0.Export = TRUE) AND (MpAlarmXHistory_0.CommandDone = TRUE)) THEN
		HmiAlarmX.Commands.ExportAlarms := FALSE;
		MpAlarmXHistory_0.Export := FALSE;
	END_IF

    // Error reset
    IF NOT MpAlarmXCore_0.Error THEN
        MpAlarmXCore_0.ErrorReset := FALSE;
    END_IF
    IF NOT MpAlarmXListUI_0.Error THEN
        MpAlarmXListUI_0.ErrorReset := FALSE;
    END_IF
    IF NOT MpAlarmXHistory_0.Error THEN
        MpAlarmXHistory_0.ErrorReset := FALSE;
    END_IF
    IF NOT MpAlarmXHistoryUI_0.Error THEN
        MpAlarmXHistoryUI_0.ErrorReset := FALSE;
    END_IF

	// Assign MpLinks & UIConnects
	MpAlarmXCore_0.MpLink := ADR(gMpLinkAlarmXCore);
	MpAlarmXListUI_0.MpLink := ADR(gMpLinkAlarmXCore);
	MpAlarmXListUI_0.UIConnect := ADR(MpAlarmXListUIConnect);
	MpAlarmXHistory_0.MpLink := ADR(gMpLinkAlarmXHistory);
	MpAlarmXHistoryUI_0.MpLink := ADR(gMpLinkAlarmXHistory);
	MpAlarmXHistoryUI_0.UIConnect := ADR(MpAlarmXHistoryUIConnect);

	// Call function blocks
	MpAlarmXCore_0();
	MpAlarmXListUI_0();
	MpAlarmXHistory_0();
	MpAlarmXHistoryUI_0();

END_PROGRAM

PROGRAM _EXIT

	// Disable the function blocls to unlink the MpLinks
    MpAlarmXCore_0.Enable := FALSE;
    MpAlarmXListUI_0.Enable := FALSE;
    MpAlarmXHistory_0.Enable := FALSE;
	MpAlarmXHistoryUI_0.Enable := FALSE;
	QueryActiveAlarms.Enable := FALSE;

	// Call function blocks
    MpAlarmXCore_0();
    MpAlarmXListUI_0();
    MpAlarmXHistory_0();
    MpAlarmXHistoryUI_0();
    QueryActiveAlarms();

END_PROGRAM
```

### Program Logical/Infrastructure/AlarmX/AlarmMgt (IEC)
